LIN {X 0,Y 397.717,Z 584.928,A -85,B 0,C 180,E1 -19257.729,E2 -19257.729} C_VEL
LIN {X 0,Y 395.996,Z 592.127,A -85,B 0,C 180,E1 -19259.493,E2 -19259.493} C_VEL
LIN {X 0,Y 394.774,Z 597.161,A -85,B 0,C 180,E1 -19261.017,E2 -19261.017} C_VEL
LIN {X 0,Y 393.567,Z 602.32,A -85,B 0,C 180,E1 -19263.061,E2 -19263.061} C_VEL
LIN {X 0,Y 392.834,Z 605.925,A -85,B 0,C 180,E1 -19265.115,E2 -19265.115} C_VEL
LIN {X 0,Y 392.166,Z 608.094,A -85,B 0,C 180,E1 -19267.182,E2 -19267.182} C_VEL
LIN {X 0,Y 391.836,Z 608.822,A -85,B 0,C 180,E1 -19269.258,E2 -19269.258} C_VEL
LIN {X 0,Y 391.759,Z 608.57,A -85,B 0,C 180,E1 -19270.455,E2 -19270.455} C_VEL
LIN {X 0,Y 391.593,Z 607.122,A -85,B 0,C 180,E1 -19272.395,E2 -19272.395} C_VEL
LIN {X 0,Y 391.705,Z 604.06,A -85,B 0,C 180,E1 -19274.498,E2 -19274.498} C_VEL
LIN {X 0,Y 391.827,Z 600.696,A -85,B 0,C 180,E1 -19276.086,E2 -19276.086} C_VEL
LIN {X 0,Y 392.017,Z 596.311,A -85,B 0,C 180,E1 -19277.683,E2 -19277.683} C_VEL
LIN {X 0,Y 392.321,Z 589.701,A -85,B 0,C 180,E1 -19279.558,E2 -19279.558} C_VEL
LIN {X 0,Y 392.753,Z 582.648,A -85,B 0,C 180,E1 -19281.17,E2 -19281.17} C_VEL
LIN {X 0,Y 393.306,Z 574.032,A -85,B 0,C 180,E1 -19282.789,E2 -19282.789} C_VEL
LIN {X 0,Y 394.075,Z 563.557,A -85,B 0,C 180,E1 -19284.406,E2 -19284.406} C_VEL
LIN {X 0,Y 394.825,Z 552.905,A -85,B 0,C 180,E1 -19285.763,E2 -19285.763} C_VEL
LIN {X 0,Y 395.691,Z 541.405,A -85,B 0,C 180,E1 -19286.975,E2 -19286.975} C_VEL
LIN {X 0,Y 396.569,Z 527.738,A -85,B 0,C 180,E1 -19288.141,E2 -19288.141} C_VEL
LIN {X 0,Y 397.394,Z 514.095,A -85,B 0,C 180,E1 -19289.066,E2 -19289.066} C_VEL
LIN {X 0,Y 398.175,Z 500.064,A -85,B 0,C 180,E1 -19289.799,E2 -19289.799} C_VEL
LIN {X 0,Y 398.925,Z 485.084,A -85,B 0,C 180,E1 -19290.355,E2 -19290.355} C_VEL
LIN {X 0,Y 400.788,Z 412.237,A -85,B 0,C 180,E1 -19292.1,E2 -19292.1} C_VEL
LIN {X 0,Y 401.807,Z 378.965,A -85,B 0,C 180,E1 -19292.889,E2 -19292.889} C_VEL
LIN {X 0,Y 397.729,Z 345.32,A -85,B 0,C 180,E1 -19293.857,E2 -19293.857} C_VEL
LIN {X 0,Y 397.72,Z 344.139,A -85,B 0,C 180,E1 -19293.988,E2 -19293.988} C_VEL
LIN {X 0,Y 398.553,Z 329.713,A -85,B 0,C 180,E1 -19296.319,E2 -19296.319} C_VEL
LIN {X 0,Y 395.358,Z 313.634,A -85,B 0,C 180,E1 -19299.097,E2 -19299.097} C_VEL
LIN {X 0,Y 394.215,Z 307.939,A -85,B 0,C 180,E1 -19300.103,E2 -19300.103} C_VEL
LIN {X 0,Y 394.182,Z 307.94,A -85,B 0,C 180,E1 -19303.869,E2 -19303.869} C_VEL
LIN {X 0,Y 394.119,Z 307.946,A -85,B 0,C 180,E1 -19307.516,E2 -19307.516} C_VEL
LIN {X 0,Y 394.135,Z 307.949,A -85,B 0,C 180,E1 -19310.222,E2 -19310.222} C_VEL
LIN {X 0,Y 394.157,Z 307.941,A -85,B 0,C 180,E1 -19313.1,E2 -19313.1} C_VEL
LIN {X 0,Y 394.182,Z 307.939,A -85,B 0,C 180,E1 -19316.572,E2 -19316.572} C_VEL
LIN {X 0,Y 394.175,Z 307.944,A -85,B 0,C 180,E1 -19320.159,E2 -19320.159} C_VEL
LIN {X 0,Y 394.204,Z 307.936,A -85,B 0,C 180,E1 -19323.625,E2 -19323.625} C_VEL
LIN {X 0,Y 394.26,Z 307.93,A -85,B 0,C 180,E1 -19327.493,E2 -19327.493} C_VEL
LIN {X 0,Y 394.254,Z 307.93,A -85,B 0,C 180,E1 -19331.347,E2 -19331.347} C_VEL
LIN {X 0,Y 394.308,Z 307.924,A -85,B 0,C 180,E1 -19334.544,E2 -19334.544} C_VEL
LIN {X 0,Y 394.417,Z 307.915,A -85,B 0,C 180,E1 -19337.693,E2 -19337.693} C_VEL
LIN {X 0,Y 394.399,Z 308.039,A -85,B 0,C 180,E1 -19338.871,E2 -19338.871} C_VEL
LIN {X 0,Y 394.702,Z 309.634,A -85,B 0,C 180,E1 -19339.279,E2 -19339.279} C_VEL
LIN {X 0,Y 403.21,Z 335.163,A -85,B 0,C 180,E1 -19340.175,E2 -19340.175} C_VEL
LIN {X 0,Y 403.99,Z 339.498,A -85,B 0,C 180,E1 -19340.292,E2 -19340.292} C_VEL
LIN {X 0,Y 401.838,Z 445.209,A -85,B 0,C 180,E1 -19342.171,E2 -19342.171} C_VEL
LIN {X 0,Y 401.351,Z 459.684,A -85,B 0,C 180,E1 -19342.634,E2 -19342.634} C_VEL
LIN {X 0,Y 400.697,Z 473.526,A -85,B 0,C 180,E1 -19343.284,E2 -19343.284} C_VEL
LIN {X 0,Y 399.792,Z 486.451,A -85,B 0,C 180,E1 -19344.09,E2 -19344.09} C_VEL
LIN {X 0,Y 398.99,Z 497.538,A -85,B 0,C 180,E1 -19344.962,E2 -19344.962} C_VEL
LIN {X 0,Y 397.656,Z 509.289,A -85,B 0,C 180,E1 -19346.084,E2 -19346.084} C_VEL
LIN {X 0,Y 396.813,Z 518.984,A -85,B 0,C 180,E1 -19347.215,E2 -19347.215} C_VEL
LIN {X 0,Y 395.904,Z 528.108,A -85,B 0,C 180,E1 -19348.477,E2 -19348.477} C_VEL
LIN {X 0,Y 394.823,Z 537.282,A -85,B 0,C 180,E1 -19349.998,E2 -19349.998} C_VEL
LIN {X 0,Y 394.061,Z 544.913,A -85,B 0,C 180,E1 -19351.525,E2 -19351.525} C_VEL
LIN {X 0,Y 393.463,Z 551.26,A -85,B 0,C 180,E1 -19353.059,E2 -19353.059} C_VEL
LIN {X 0,Y 393.104,Z 556.487,A -85,B 0,C 180,E1 -19354.596,E2 -19354.596} C_VEL
LIN {X 0,Y 392.549,Z 562.047,A -85,B 0,C 180,E1 -19356.658,E2 -19356.658} C_VEL
LIN {X 0,Y 392.238,Z 565.16,A -85,B 0,C 180,E1 -19358.211,E2 -19358.211} C_VEL
LIN {X 0,Y 392.167,Z 568.068,A -85,B 0,C 180,E1 -19360.286,E2 -19360.286} C_VEL
LIN {X 0,Y 392.135,Z 569.619,A -85,B 0,C 180,E1 -19362.375,E2 -19362.375} C_VEL
LIN {X 0,Y 392.357,Z 569.815,A -85,B 0,C 180,E1 -19364.471,E2 -19364.471} C_VEL
LIN {X 0,Y 392.721,Z 568.654,A -85,B 0,C 180,E1 -19366.578,E2 -19366.578} C_VEL
LIN {X 0,Y 393.38,Z 566.06,A -85,B 0,C 180,E1 -19368.69,E2 -19368.69} C_VEL
LIN {X 0,Y 394.327,Z 561.953,A -85,B 0,C 180,E1 -19370.806,E2 -19370.806} C_VEL
LIN {X 0,Y 395.598,Z 556.204,A -85,B 0,C 180,E1 -19372.922,E2 -19372.922} C_VEL
LIN {X 0,Y 397.028,Z 549.645,A -85,B 0,C 180,E1 -19374.768,E2 -19374.768} C_VEL
LIN {X 0,Y 398.559,Z 542.753,A -85,B 0,C 180,E1 -19376.325,E2 -19376.325} C_VEL
LIN {X 0,Y 400.232,Z 534.249,A -85,B 0,C 180,E1 -19377.911,E2 -19377.911} C_VEL
LIN {X 0,Y 402.147,Z 524.22,A -85,B 0,C 180,E1 -19379.439,E2 -19379.439} C_VEL
LIN {X 0,Y 403.955,Z 513.61,A -85,B 0,C 180,E1 -19380.762,E2 -19380.762} C_VEL
LIN {X 0,Y 405.704,Z 502.263,A -85,B 0,C 180,E1 -19381.917,E2 -19381.917} C_VEL
LIN {X 0,Y 407.33,Z 489.783,A -85,B 0,C 180,E1 -19382.94,E2 -19382.94} C_VEL
LIN {X 0,Y 408.67,Z 476.909,A -85,B 0,C 180,E1 -19383.774,E2 -19383.774} C_VEL
LIN {X 0,Y 409.658,Z 464.519,A -85,B 0,C 180,E1 -19384.393,E2 -19384.393} C_VEL
LIN {X 0,Y 409.957,Z 460.294,A -85,B 0,C 180,E1 -19384.563,E2 -19384.563} C_VEL
LIN {X 0,Y 409.856,Z 454.652,A -85,B 0,C 180,E1 -19384.802,E2 -19384.802} C_VEL
LIN {X 0,Y 407.721,Z 445.503,A -85,B 0,C 180,E1 -19385.244,E2 -19385.244} C_VEL
LIN {X 0,Y 405.273,Z 436.264,A -85,B 0,C 180,E1 -19385.632,E2 -19385.632} C_VEL
LIN {X 0,Y 404.725,Z 430.471,A -85,B 0,C 180,E1 -19385.789,E2 -19385.789} C_VEL
LIN {X 0,Y 407.027,Z 352.192,A -85,B 0,C 180,E1 -19387.172,E2 -19387.172} C_VEL
LIN {X 0,Y 399.145,Z 334.318,A -85,B 0,C 180,E1 -19388.191,E2 -19388.191} C_VEL
LIN {X 0,Y 390.851,Z 317.809,A -85,B 0,C 180,E1 -19389.271,E2 -19389.271} C_VEL
LIN {X 0,Y 387.76,Z 311.713,A -85,B 0,C 180,E1 -19389.72,E2 -19389.72} C_VEL
LIN {X 0,Y 387.081,Z 308.822,A -85,B 0,C 180,E1 -19390.646,E2 -19390.646} C_VEL
LIN {X 0,Y 387.096,Z 308.822,A -85,B 0,C 180,E1 -19393.631,E2 -19393.631} C_VEL
LIN {X 0,Y 387.087,Z 308.827,A -85,B 0,C 180,E1 -19396.558,E2 -19396.558} C_VEL
LIN {X 0,Y 387.084,Z 308.827,A -85,B 0,C 180,E1 -19399.46,E2 -19399.46} C_VEL
LIN {X 0,Y 387.129,Z 308.809,A -85,B 0,C 180,E1 -19402.754,E2 -19402.754} C_VEL
LIN {X 0,Y 387.132,Z 308.804,A -85,B 0,C 180,E1 -19405.883,E2 -19405.883} C_VEL
LIN {X 0,Y 387.133,Z 308.813,A -85,B 0,C 180,E1 -19409.562,E2 -19409.562} C_VEL
LIN {X 0,Y 387.145,Z 308.807,A -85,B 0,C 180,E1 -19413.108,E2 -19413.108} C_VEL
LIN {X 0,Y 387.133,Z 308.818,A -85,B 0,C 180,E1 -19415.409,E2 -19415.409} C_VEL
LIN {X 0,Y 387.191,Z 308.806,A -85,B 0,C 180,E1 -19417.673,E2 -19417.673} C_VEL
LIN {X 0,Y 387.177,Z 308.802,A -85,B 0,C 180,E1 -19420.996,E2 -19420.996} C_VEL
LIN {X 0,Y 387.194,Z 308.809,A -85,B 0,C 180,E1 -19424.255,E2 -19424.255} C_VEL
LIN {X 0,Y 387.311,Z 308.795,A -85,B 0,C 180,E1 -19427.559,E2 -19427.559} C_VEL
LIN {X 0,Y 387.371,Z 308.778,A -85,B 0,C 180,E1 -19431.683,E2 -19431.683} C_VEL
LIN {X 0,Y 387.458,Z 308.776,A -85,B 0,C 180,E1 -19434.814,E2 -19434.814} C_VEL
LIN {X 0,Y 387.4,Z 308.783,A -85,B 0,C 180,E1 -19437.928,E2 -19437.928} C_VEL
LIN {X 0,Y 387.389,Z 308.774,A -85,B 0,C 180,E1 -19441.036,E2 -19441.036} C_VEL
LIN {X 0,Y 387.498,Z 308.771,A -85,B 0,C 180,E1 -19444.146,E2 -19444.146} C_VEL
LIN {X 0,Y 387.402,Z 308.768,A -85,B 0,C 180,E1 -19447.271,E2 -19447.271} C_VEL
LIN {X 0,Y 387.311,Z 308.795,A -85,B 0,C 180,E1 -19450.419,E2 -19450.419} C_VEL
LIN {X 0,Y 387.345,Z 308.775,A -85,B 0,C 180,E1 -19452.533,E2 -19452.533} C_VEL
LIN {X 0,Y 387.248,Z 308.794,A -85,B 0,C 180,E1 -19456.546,E2 -19456.546} C_VEL
LIN {X 0,Y 387.191,Z 308.81,A -85,B 0,C 180,E1 -19460.104,E2 -19460.104} C_VEL
LIN {X 0,Y 387.144,Z 308.815,A -85,B 0,C 180,E1 -19463.456,E2 -19463.456} C_VEL
LIN {X 0,Y 387.145,Z 308.812,A -85,B 0,C 180,E1 -19465.736,E2 -19465.736} C_VEL
LIN {X 0,Y 387.15,Z 308.814,A -85,B 0,C 180,E1 -19469.242,E2 -19469.242} C_VEL
LIN {X 0,Y 387.132,Z 308.817,A -85,B 0,C 180,E1 -19472.874,E2 -19472.874} C_VEL
LIN {X 0,Y 387.198,Z 308.781,A -85,B 0,C 180,E1 -19476.654,E2 -19476.654} C_VEL
LIN {X 0,Y 387.15,Z 308.816,A -85,B 0,C 180,E1 -19479.289,E2 -19479.289} C_VEL
LIN {X 0,Y 387.107,Z 308.823,A -85,B 0,C 180,E1 -19482.114,E2 -19482.114} C_VEL
LIN {X 0,Y 387.143,Z 308.813,A -85,B 0,C 180,E1 -19485.125,E2 -19485.125} C_VEL
LIN {X 0,Y 387.139,Z 308.818,A -85,B 0,C 180,E1 -19487.981,E2 -19487.981} C_VEL
LIN {X 0,Y 387.163,Z 308.815,A -85,B 0,C 180,E1 -19491.073,E2 -19491.073} C_VEL
LIN {X 0,Y 387.226,Z 308.853,A -85,B 0,C 180,E1 -19493.089,E2 -19493.089} C_VEL
LIN {X 0,Y 390.309,Z 320.663,A -85,B 0,C 180,E1 -19496.202,E2 -19496.202} C_VEL
LIN {X 0,Y 392.504,Z 330.055,A -85,B 0,C 180,E1 -19498.538,E2 -19498.538} C_VEL
LIN {X 0,Y 395.104,Z 342.29,A -85,B 0,C 180,E1 -19501.406,E2 -19501.406} C_VEL
LIN {X 0,Y 395.811,Z 345.929,A -85,B 0,C 180,E1 -19502.23,E2 -19502.23} C_VEL
LIN {X 0,Y 395.398,Z 349.986,A -85,B 0,C 180,E1 -19503.051,E2 -19503.051} C_VEL
LIN {X 0,Y 401.869,Z 383.713,A -85,B 0,C 180,E1 -19504.294,E2 -19504.294} C_VEL
LIN {X 0,Y 405.569,Z 408.629,A -85,B 0,C 180,E1 -19505.089,E2 -19505.089} C_VEL
LIN {X 0,Y 403.302,Z 488.379,A -85,B 0,C 180,E1 -19506.527,E2 -19506.527} C_VEL
LIN {X 0,Y 402.306,Z 502.975,A -85,B 0,C 180,E1 -19506.974,E2 -19506.974} C_VEL
LIN {X 0,Y 400.773,Z 516.935,A -85,B 0,C 180,E1 -19507.593,E2 -19507.593} C_VEL
LIN {X 0,Y 399.336,Z 528.164,A -85,B 0,C 180,E1 -19508.254,E2 -19508.254} C_VEL
LIN {X 0,Y 397.405,Z 540.887,A -85,B 0,C 180,E1 -19509.207,E2 -19509.207} C_VEL
LIN {X 0,Y 395.458,Z 552.842,A -85,B 0,C 180,E1 -19510.337,E2 -19510.337} C_VEL
LIN {X 0,Y 393.385,Z 563.621,A -85,B 0,C 180,E1 -19511.579,E2 -19511.579} C_VEL
LIN {X 0,Y 391.238,Z 574.311,A -85,B 0,C 180,E1 -19513.089,E2 -19513.089} C_VEL
LIN {X 0,Y 389.501,Z 583.171,A -85,B 0,C 180,E1 -19514.621,E2 -19514.621} C_VEL
LIN {X 0,Y 387.915,Z 591.702,A -85,B 0,C 180,E1 -19516.427,E2 -19516.427} C_VEL
LIN {X 0,Y 386.65,Z 598.451,A -85,B 0,C 180,E1 -19518.196,E2 -19518.196} C_VEL
LIN {X 0,Y 385.7,Z 604.145,A -85,B 0,C 180,E1 -19520.068,E2 -19520.068} C_VEL
LIN {X 0,Y 385.045,Z 608.993,A -85,B 0,C 180,E1 -19522.161,E2 -19522.161} C_VEL
LIN {X 0,Y 384.927,Z 612.688,A -85,B 0,C 180,E1 -19524.521,E2 -19524.521} C_VEL
LIN {X 0,Y 384.895,Z 613.051,A -85,B 0,C 180,E1 -19524.782,E2 -19524.782} C_VEL
LIN {X 0,Y 384.85,Z 617.082,A -85,B 0,C 180,E1 -19526.35,E2 -19526.35} C_VEL
LIN {X 0,Y 384.85,Z 620.126,A -85,B 0,C 180,E1 -19527.916,E2 -19527.916} C_VEL
LIN {X 0,Y 384.897,Z 621.672,A -85,B 0,C 180,E1 -19528.96,E2 -19528.96} C_VEL
LIN {X 0,Y 384.811,Z 623.592,A -85,B 0,C 180,E1 -19531.045,E2 -19531.045} C_VEL
LIN {X 0,Y 384.734,Z 624.032,A -85,B 0,C 180,E1 -19533.133,E2 -19533.133} C_VEL
LIN {X 0,Y 384.873,Z 623.036,A -85,B 0,C 180,E1 -19535.223,E2 -19535.223} C_VEL
LIN {X 0,Y 385.213,Z 620.617,A -85,B 0,C 180,E1 -19537.315,E2 -19537.315} C_VEL
LIN {X 0,Y 385.94,Z 616.726,A -85,B 0,C 180,E1 -19539.403,E2 -19539.403} C_VEL
LIN {X 0,Y 387.261,Z 611.271,A -85,B 0,C 180,E1 -19541.478,E2 -19541.478} C_VEL
LIN {X 0,Y 388.362,Z 605.739,A -85,B 0,C 180,E1 -19543.11,E2 -19543.11} C_VEL
LIN {X 0,Y 390.047,Z 598.548,A -85,B 0,C 180,E1 -19544.829,E2 -19544.829} C_VEL
LIN {X 0,Y 392.246,Z 589.302,A -85,B 0,C 180,E1 -19546.604,E2 -19546.604} C_VEL
LIN {X 0,Y 394.204,Z 579.747,A -85,B 0,C 180,E1 -19548.119,E2 -19548.119} C_VEL
LIN {X 0,Y 396.511,Z 569.228,A -85,B 0,C 180,E1 -19549.479,E2 -19549.479} C_VEL
LIN {X 0,Y 398.985,Z 556.544,A -85,B 0,C 180,E1 -19550.826,E2 -19550.826} C_VEL
LIN {X 0,Y 401.271,Z 543.87,A -85,B 0,C 180,E1 -19551.91,E2 -19551.91} C_VEL
LIN {X 0,Y 403.32,Z 530.585,A -85,B 0,C 180,E1 -19552.812,E2 -19552.812} C_VEL
LIN {X 0,Y 405.461,Z 514.876,A -85,B 0,C 180,E1 -19553.616,E2 -19553.616} C_VEL
LIN {X 0,Y 407.077,Z 500.015,A -85,B 0,C 180,E1 -19554.157,E2 -19554.157} C_VEL
LIN {X 0,Y 413.308,Z 410.128,A -85,B 0,C 180,E1 -19556.57,E2 -19556.57} C_VEL
LIN {X 0,Y 412.123,Z 392.284,A -85,B 0,C 180,E1 -19557.379,E2 -19557.379} C_VEL
LIN {X 0,Y 410.315,Z 375.608,A -85,B 0,C 180,E1 -19558.261,E2 -19558.261} C_VEL
LIN {X 0,Y 407.875,Z 359.524,A -85,B 0,C 180,E1 -19559.257,E2 -19559.257} C_VEL
LIN {X 0,Y 406.787,Z 354.086,A -85,B 0,C 180,E1 -19559.649,E2 -19559.649} C_VEL
LIN {X 0,Y 405.35,Z 347.684,A -85,B 0,C 180,E1 -19560.497,E2 -19560.497} C_VEL
LIN {X 0,Y 403.914,Z 340.609,A -85,B 0,C 180,E1 -19561.527,E2 -19561.527} C_VEL
LIN {X 0,Y 402.643,Z 336.786,A -85,B 0,C 180,E1 -19562.224,E2 -19562.224} C_VEL
LIN {X 0,Y 398.176,Z 328.661,A -85,B 0,C 180,E1 -19564.26,E2 -19564.26} C_VEL
LIN {X 0,Y 394.492,Z 322.113,A -85,B 0,C 180,E1 -19566.247,E2 -19566.247} C_VEL
LIN {X 0,Y 392.786,Z 318.98,A -85,B 0,C 180,E1 -19567.326,E2 -19567.326} C_VEL
LIN {X 0,Y 390.499,Z 315.506,A -85,B 0,C 180,E1 -19568.891,E2 -19568.891} C_VEL
LIN {X 0,Y 389.955,Z 313.964,A -85,B 0,C 180,E1 -19569.432,E2 -19569.432} C_VEL
LIN {X 0,Y 387.569,Z 310.664,A -85,B 0,C 180,E1 -19571.409,E2 -19571.409} C_VEL
LIN {X 0,Y 387.099,Z 308.821,A -85,B 0,C 180,E1 -19572.381,E2 -19572.381} C_VEL
LIN {X 0,Y 387.121,Z 308.818,A -85,B 0,C 180,E1 -19575.117,E2 -19575.117} C_VEL
LIN {X 0,Y 387.098,Z 308.823,A -85,B 0,C 180,E1 -19577.971,E2 -19577.971} C_VEL
LIN {X 0,Y 387.11,Z 308.823,A -85,B 0,C 180,E1 -19581.085,E2 -19581.085} C_VEL
LIN {X 0,Y 387.174,Z 308.813,A -85,B 0,C 180,E1 -19584.625,E2 -19584.625} C_VEL
LIN {X 0,Y 387.147,Z 308.831,A -85,B 0,C 180,E1 -19586.733,E2 -19586.733} C_VEL
LIN {X 0,Y 388.13,Z 311.639,A -85,B 0,C 180,E1 -19588.443,E2 -19588.443} C_VEL
LIN {X 0,Y 389.475,Z 313.721,A -85,B 0,C 180,E1 -19589.764,E2 -19589.764} C_VEL
LIN {X 0,Y 391.233,Z 317.506,A -85,B 0,C 180,E1 -19591.647,E2 -19591.647} C_VEL
LIN {X 0,Y 393.675,Z 323.256,A -85,B 0,C 180,E1 -19594.046,E2 -19594.046} C_VEL
LIN {X 0,Y 396.597,Z 330.734,A -85,B 0,C 180,E1 -19596.696,E2 -19596.696} C_VEL
LIN {X 0,Y 398.941,Z 337.757,A -85,B 0,C 180,E1 -19598.849,E2 -19598.849} C_VEL
LIN {X 0,Y 401.343,Z 346.482,A -85,B 0,C 180,E1 -19601.22,E2 -19601.22} C_VEL
LIN {X 0,Y 401.755,Z 348.046,A -85,B 0,C 180,E1 -19601.562,E2 -19601.562} C_VEL
LIN {X 0,Y 407.126,Z 358.325,A -85,B 0,C 180,E1 -19602.857,E2 -19602.857} C_VEL
LIN {X 0,Y 410.673,Z 366.267,A -85,B 0,C 180,E1 -19603.695,E2 -19603.695} C_VEL
LIN {X 0,Y 413.329,Z 380.205,A -85,B 0,C 180,E1 -19604.595,E2 -19604.595} C_VEL
LIN {X 0,Y 414.901,Z 391.129,A -85,B 0,C 180,E1 -19605.201,E2 -19605.201} C_VEL
LIN {X 0,Y 407.833,Z 488.797,A -85,B 0,C 180,E1 -19607.792,E2 -19607.792} C_VEL
LIN {X 0,Y 406.346,Z 503.456,A -85,B 0,C 180,E1 -19608.377,E2 -19608.377} C_VEL
LIN {X 0,Y 404.584,Z 517.538,A -85,B 0,C 180,E1 -19609.148,E2 -19609.148} C_VEL
LIN {X 0,Y 402.459,Z 531.281,A -85,B 0,C 180,E1 -19610.104,E2 -19610.104} C_VEL
LIN {X 0,Y 400.294,Z 543.672,A -85,B 0,C 180,E1 -19611.193,E2 -19611.193} C_VEL
LIN {X 0,Y 397.851,Z 556.012,A -85,B 0,C 180,E1 -19612.539,E2 -19612.539} C_VEL
LIN {X 0,Y 395.719,Z 566.254,A -85,B 0,C 180,E1 -19613.903,E2 -19613.903} C_VEL
LIN {X 0,Y 393.861,Z 574.529,A -85,B 0,C 180,E1 -19615.221,E2 -19615.221} C_VEL
LIN {X 0,Y 391.606,Z 583.459,A -85,B 0,C 180,E1 -19616.924,E2 -19616.924} C_VEL
LIN {X 0,Y 389.876,Z 590.014,A -85,B 0,C 180,E1 -19618.456,E2 -19618.456} C_VEL
LIN {X 0,Y 388.079,Z 597.03,A -85,B 0,C 180,E1 -19620.517,E2 -19620.517} C_VEL
LIN {X 0,Y 387.039,Z 601.106,A -85,B 0,C 180,E1 -19622.074,E2 -19622.074} C_VEL
LIN {X 0,Y 386.112,Z 605.178,A -85,B 0,C 180,E1 -19624.161,E2 -19624.161} C_VEL
LIN {X 0,Y 385.351,Z 607.788,A -85,B 0,C 180,E1 -19626.261,E2 -19626.261} C_VEL
LIN {X 0,Y 384.833,Z 608.92,A -85,B 0,C 180,E1 -19628.373,E2 -19628.373} C_VEL
LIN {X 0,Y 384.652,Z 608.602,A -85,B 0,C 180,E1 -19630.492,E2 -19630.492} C_VEL
LIN {X 0,Y 384.504,Z 606.802,A -85,B 0,C 180,E1 -19632.627,E2 -19632.627} C_VEL
LIN {X 0,Y 384.627,Z 603.466,A -85,B 0,C 180,E1 -19634.771,E2 -19634.771} C_VEL
LIN {X 0,Y 384.772,Z 599.82,A -85,B 0,C 180,E1 -19636.389,E2 -19636.389} C_VEL
LIN {X 0,Y 384.97,Z 595.132,A -85,B 0,C 180,E1 -19638.018,E2 -19638.018} C_VEL
LIN {X 0,Y 385.334,Z 588.18,A -85,B 0,C 180,E1 -19639.927,E2 -19639.927} C_VEL
LIN {X 0,Y 385.755,Z 580.768,A -85,B 0,C 180,E1 -19641.568,E2 -19641.568} C_VEL
LIN {X 0,Y 386.378,Z 571.701,A -85,B 0,C 180,E1 -19643.222,E2 -19643.222} C_VEL
LIN {X 0,Y 387.175,Z 561.079,A -85,B 0,C 180,E1 -19644.806,E2 -19644.806} C_VEL
LIN {X 0,Y 388.055,Z 549.327,A -85,B 0,C 180,E1 -19646.246,E2 -19646.246} C_VEL
LIN {X 0,Y 388.918,Z 537.005,A -85,B 0,C 180,E1 -19647.484,E2 -19647.484} C_VEL
LIN {X 0,Y 389.774,Z 524.543,A -85,B 0,C 180,E1 -19648.504,E2 -19648.504} C_VEL
LIN {X 0,Y 390.571,Z 510.645,A -85,B 0,C 180,E1 -19649.402,E2 -19649.402} C_VEL
LIN {X 0,Y 391.353,Z 495.282,A -85,B 0,C 180,E1 -19650.15,E2 -19650.15} C_VEL
LIN {X 0,Y 391.98,Z 480.362,A -85,B 0,C 180,E1 -19650.653,E2 -19650.653} C_VEL
LIN {X 0,Y 394.773,Z 379.081,A -85,B 0,C 180,E1 -19653.104,E2 -19653.104} C_VEL
LIN {X 0,Y 390.726,Z 344.841,A -85,B 0,C 180,E1 -19654.132,E2 -19654.132} C_VEL
LIN {X 0,Y 391.585,Z 330.973,A -85,B 0,C 180,E1 -19656.393,E2 -19656.393} C_VEL
LIN {X 0,Y 388.442,Z 315.155,A -85,B 0,C 180,E1 -19659.158,E2 -19659.158} C_VEL
LIN {X 0,Y 387.138,Z 308.822,A -85,B 0,C 180,E1 -19660.292,E2 -19660.292} C_VEL
LIN {X 0,Y 387.119,Z 308.819,A -85,B 0,C 180,E1 -19663.632,E2 -19663.632} C_VEL
LIN {X 0,Y 387.083,Z 308.827,A -85,B 0,C 180,E1 -19666.555,E2 -19666.555} C_VEL
LIN {X 0,Y 387.096,Z 308.82,A -85,B 0,C 180,E1 -19669.463,E2 -19669.463} C_VEL
LIN {X 0,Y 387.131,Z 308.818,A -85,B 0,C 180,E1 -19672.759,E2 -19672.759} C_VEL
LIN {X 0,Y 387.118,Z 308.819,A -85,B 0,C 180,E1 -19676.337,E2 -19676.337} C_VEL
LIN {X 0,Y 387.126,Z 308.818,A -85,B 0,C 180,E1 -19679.559,E2 -19679.559} C_VEL
LIN {X 0,Y 387.154,Z 308.812,A -85,B 0,C 180,E1 -19683.106,E2 -19683.106} C_VEL
LIN {X 0,Y 387.14,Z 308.816,A -85,B 0,C 180,E1 -19685.407,E2 -19685.407} C_VEL
LIN {X 0,Y 387.218,Z 308.809,A -85,B 0,C 180,E1 -19687.672,E2 -19687.672} C_VEL
LIN {X 0,Y 387.208,Z 308.807,A -85,B 0,C 180,E1 -19690.995,E2 -19690.995} C_VEL
LIN {X 0,Y 387.267,Z 308.804,A -85,B 0,C 180,E1 -19694.256,E2 -19694.256} C_VEL
LIN {X 0,Y 387.34,Z 308.796,A -85,B 0,C 180,E1 -19697.556,E2 -19697.556} C_VEL
LIN {X 0,Y 387.357,Z 308.885,A -85,B 0,C 180,E1 -19698.623,E2 -19698.623} C_VEL
LIN {X 0,Y 387.566,Z 310.046,A -85,B 0,C 180,E1 -19698.924,E2 -19698.924} C_VEL
LIN {X 0,Y 396.649,Z 337.095,A -85,B 0,C 180,E1 -19699.9,E2 -19699.9} C_VEL
LIN {X 0,Y 397.206,Z 339.535,A -85,B 0,C 180,E1 -19699.972,E2 -19699.972} C_VEL
LIN {X 0,Y 395.021,Z 446.166,A -85,B 0,C 180,E1 -19701.907,E2 -19701.907} C_VEL
LIN {X 0,Y 394.514,Z 460.458,A -85,B 0,C 180,E1 -19702.377,E2 -19702.377} C_VEL
LIN {X 0,Y 393.847,Z 474.202,A -85,B 0,C 180,E1 -19703.039,E2 -19703.039} C_VEL
LIN {X 0,Y 392.91,Z 487.072,A -85,B 0,C 180,E1 -19703.857,E2 -19703.857} C_VEL
LIN {X 0,Y 392.048,Z 498.129,A -85,B 0,C 180,E1 -19704.744,E2 -19704.744} C_VEL
LIN {X 0,Y 390.731,Z 509.837,A -85,B 0,C 180,E1 -19705.886,E2 -19705.886} C_VEL
LIN {X 0,Y 389.786,Z 520.471,A -85,B 0,C 180,E1 -19707.165,E2 -19707.165} C_VEL
LIN {X 0,Y 388.804,Z 529.429,A -85,B 0,C 180,E1 -19708.449,E2 -19708.449} C_VEL
LIN {X 0,Y 387.744,Z 538.445,A -85,B 0,C 180,E1 -19709.997,E2 -19709.997} C_VEL
LIN {X 0,Y 386.9,Z 545.956,A -85,B 0,C 180,E1 -19711.554,E2 -19711.554} C_VEL
LIN {X 0,Y 386.398,Z 552.209,A -85,B 0,C 180,E1 -19713.115,E2 -19713.115} C_VEL
LIN {X 0,Y 385.986,Z 557.355,A -85,B 0,C 180,E1 -19714.681,E2 -19714.681} C_VEL
LIN {X 0,Y 385.557,Z 561.561,A -85,B 0,C 180,E1 -19716.255,E2 -19716.255} C_VEL
LIN {X 0,Y 385.143,Z 565.827,A -85,B 0,C 180,E1 -19718.363,E2 -19718.363} C_VEL
LIN {X 0,Y 385.081,Z 568.644,A -85,B 0,C 180,E1 -19720.477,E2 -19720.477} C_VEL
LIN {X 0,Y 385.069,Z 570.106,A -85,B 0,C 180,E1 -19722.605,E2 -19722.605} C_VEL
LIN {X 0,Y 385.304,Z 570.209,A -85,B 0,C 180,E1 -19724.741,E2 -19724.741} C_VEL
LIN {X 0,Y 385.711,Z 568.928,A -85,B 0,C 180,E1 -19726.888,E2 -19726.888} C_VEL
LIN {X 0,Y 386.429,Z 566.227,A -85,B 0,C 180,E1 -19729.04,E2 -19729.04} C_VEL
LIN {X 0,Y 387.474,Z 562.018,A -85,B 0,C 180,E1 -19731.192,E2 -19731.192} C_VEL
LIN {X 0,Y 388.815,Z 556.161,A -85,B 0,C 180,E1 -19733.346,E2 -19733.346} C_VEL
LIN {X 0,Y 390.336,Z 549.486,A -85,B 0,C 180,E1 -19735.222,E2 -19735.222} C_VEL
LIN {X 0,Y 392.156,Z 541.35,A -85,B 0,C 180,E1 -19737.034,E2 -19737.034} C_VEL
LIN {X 0,Y 394.06,Z 532.196,A -85,B 0,C 180,E1 -19738.677,E2 -19738.677} C_VEL
LIN {X 0,Y 396.164,Z 521.352,A -85,B 0,C 180,E1 -19740.254,E2 -19740.254} C_VEL
LIN {X 0,Y 398.065,Z 510.297,A -85,B 0,C 180,E1 -19741.563,E2 -19741.563} C_VEL
LIN {X 0,Y 399.77,Z 499.188,A -85,B 0,C 180,E1 -19742.637,E2 -19742.637} C_VEL
LIN {X 0,Y 401.385,Z 486.322,A -85,B 0,C 180,E1 -19743.642,E2 -19743.642} C_VEL
LIN {X 0,Y 402.69,Z 472.317,A -85,B 0,C 180,E1 -19744.496,E2 -19744.496} C_VEL
LIN {X 0,Y 403.755,Z 458.331,A -85,B 0,C 180,E1 -19745.107,E2 -19745.107} C_VEL
LIN {X 0,Y 404.44,Z 444.533,A -85,B 0,C 180,E1 -19745.513,E2 -19745.513} C_VEL
LIN {X 0,Y 404.725,Z 430.471,A -85,B 0,C 180,E1 -19745.789,E2 -19745.789} C_VEL
LIN {X 0,Y 404.266,Z 424.679,A -85,B 0,C 180,E1 -19745.939,E2 -19745.939} C_VEL
LIN {X 0,Y 399.912,Z 406.019,A -85,B 0,C 180,E1 -19746.658,E2 -19746.658} C_VEL
LIN {X 0,Y 399.426,Z 400.229,A -85,B 0,C 180,E1 -19746.815,E2 -19746.815} C_VEL
LIN {X 0,Y 400.821,Z 354.039,A -85,B 0,C 180,E1 -19747.644,E2 -19747.644} C_VEL
LIN {X 0,Y 393.009,Z 336.465,A -85,B 0,C 180,E1 -19748.68,E2 -19748.68} C_VEL
LIN {X 0,Y 384.345,Z 319.332,A -85,B 0,C 180,E1 -19749.846,E2 -19749.846} C_VEL
LIN {X 0,Y 380.665,Z 312.27,A -85,B 0,C 180,E1 -19750.375,E2 -19750.375} C_VEL
LIN {X 0,Y 380.012,Z 309.697,A -85,B 0,C 180,E1 -19751.232,E2 -19751.232} C_VEL
LIN {X 0,Y 380.054,Z 309.687,A -85,B 0,C 180,E1 -19754.45,E2 -19754.45} C_VEL
LIN {X 0,Y 380.022,Z 309.704,A -85,B 0,C 180,E1 -19757.494,E2 -19757.494} C_VEL
LIN {X 0,Y 380.056,Z 309.701,A -85,B 0,C 180,E1 -19761.199,E2 -19761.199} C_VEL
LIN {X 0,Y 380.082,Z 309.667,A -85,B 0,C 180,E1 -19764.175,E2 -19764.175} C_VEL
LIN {X 0,Y 380.075,Z 309.7,A -85,B 0,C 180,E1 -19767.694,E2 -19767.694} C_VEL
LIN {X 0,Y 380.114,Z 309.693,A -85,B 0,C 180,E1 -19770.163,E2 -19770.163} C_VEL
LIN {X 0,Y 380.093,Z 309.692,A -85,B 0,C 180,E1 -19773.751,E2 -19773.751} C_VEL
LIN {X 0,Y 380.117,Z 309.682,A -85,B 0,C 180,E1 -19777.234,E2 -19777.234} C_VEL
LIN {X 0,Y 380.141,Z 309.68,A -85,B 0,C 180,E1 -19780.63,E2 -19780.63} C_VEL
LIN {X 0,Y 380.157,Z 309.687,A -85,B 0,C 180,E1 -19783.956,E2 -19783.956} C_VEL
LIN {X 0,Y 380.268,Z 309.67,A -85,B 0,C 180,E1 -19787.471,E2 -19787.471} C_VEL
LIN {X 0,Y 380.319,Z 309.655,A -85,B 0,C 180,E1 -19791.527,E2 -19791.527} C_VEL
LIN {X 0,Y 380.409,Z 309.655,A -85,B 0,C 180,E1 -19794.718,E2 -19794.718} C_VEL
LIN {X 0,Y 380.378,Z 309.658,A -85,B 0,C 180,E1 -19797.889,E2 -19797.889} C_VEL
LIN {X 0,Y 380.356,Z 309.649,A -85,B 0,C 180,E1 -19801.055,E2 -19801.055} C_VEL
LIN {X 0,Y 380.467,Z 309.647,A -85,B 0,C 180,E1 -19804.223,E2 -19804.223} C_VEL
LIN {X 0,Y 380.357,Z 309.645,A -85,B 0,C 180,E1 -19807.407,E2 -19807.407} C_VEL
LIN {X 0,Y 380.261,Z 309.673,A -85,B 0,C 180,E1 -19810.615,E2 -19810.615} C_VEL
LIN {X 0,Y 380.279,Z 309.655,A -85,B 0,C 180,E1 -19812.77,E2 -19812.77} C_VEL
LIN {X 0,Y 380.204,Z 309.677,A -85,B 0,C 180,E1 -19816.042,E2 -19816.042} C_VEL
LIN {X 0,Y 380.162,Z 309.685,A -85,B 0,C 180,E1 -19820.014,E2 -19820.014} C_VEL
LIN {X 0,Y 380.102,Z 309.692,A -85,B 0,C 180,E1 -19823.917,E2 -19823.917} C_VEL
LIN {X 0,Y 380.126,Z 309.688,A -85,B 0,C 180,E1 -19827.43,E2 -19827.43} C_VEL
LIN {X 0,Y 380.084,Z 309.691,A -85,B 0,C 180,E1 -19831.065,E2 -19831.065} C_VEL
LIN {X 0,Y 380.1,Z 309.664,A -85,B 0,C 180,E1 -19834.839,E2 -19834.839} C_VEL
LIN {X 0,Y 380.164,Z 309.675,A -85,B 0,C 180,E1 -19837.608,E2 -19837.608} C_VEL
LIN {X 0,Y 380.057,Z 309.699,A -85,B 0,C 180,E1 -19840.925,E2 -19840.925} C_VEL
LIN {X 0,Y 380.105,Z 309.694,A -85,B 0,C 180,E1 -19844.447,E2 -19844.447} C_VEL
LIN {X 0,Y 380.085,Z 309.694,A -85,B 0,C 180,E1 -19847.489,E2 -19847.489} C_VEL
LIN {X 0,Y 380.114,Z 309.693,A -85,B 0,C 180,E1 -19851.21,E2 -19851.21} C_VEL
LIN {X 0,Y 380.166,Z 309.778,A -85,B 0,C 180,E1 -19852.492,E2 -19852.492} C_VEL
LIN {X 0,Y 383.099,Z 320.722,A -85,B 0,C 180,E1 -19855.477,E2 -19855.477} C_VEL
LIN {X 0,Y 385.643,Z 331.469,A -85,B 0,C 180,E1 -19858.219,E2 -19858.219} C_VEL
LIN {X 0,Y 388.238,Z 343.647,A -85,B 0,C 180,E1 -19861.148,E2 -19861.148} C_VEL
LIN {X 0,Y 388.994,Z 347.723,A -85,B 0,C 180,E1 -19862.088,E2 -19862.088} C_VEL
LIN {X 0,Y 388.884,Z 349.574,A -85,B 0,C 180,E1 -19862.476,E2 -19862.476} C_VEL
LIN {X 0,Y 395.239,Z 382.327,A -85,B 0,C 180,E1 -19863.718,E2 -19863.718} C_VEL
LIN {X 0,Y 399.251,Z 408.824,A -85,B 0,C 180,E1 -19864.593,E2 -19864.593} C_VEL
LIN {X 0,Y 397.589,Z 469.051,A -85,B 0,C 180,E1 -19865.685,E2 -19865.685} C_VEL
LIN {X 0,Y 396.883,Z 490.656,A -85,B 0,C 180,E1 -19866.124,E2 -19866.124} C_VEL
LIN {X 0,Y 395.732,Z 505.104,A -85,B 0,C 180,E1 -19866.603,E2 -19866.603} C_VEL
LIN {X 0,Y 394.085,Z 518.965,A -85,B 0,C 180,E1 -19867.261,E2 -19867.261} C_VEL
LIN {X 0,Y 392.298,Z 532.21,A -85,B 0,C 180,E1 -19868.114,E2 -19868.114} C_VEL
LIN {X 0,Y 390.529,Z 542.92,A -85,B 0,C 180,E1 -19868.982,E2 -19868.982} C_VEL
LIN {X 0,Y 388.339,Z 555.434,A -85,B 0,C 180,E1 -19870.236,E2 -19870.236} C_VEL
LIN {X 0,Y 386.284,Z 565.708,A -85,B 0,C 180,E1 -19871.502,E2 -19871.502} C_VEL
LIN {X 0,Y 384.091,Z 575.976,A -85,B 0,C 180,E1 -19873.038,E2 -19873.038} C_VEL
LIN {X 0,Y 382.361,Z 584.494,A -85,B 0,C 180,E1 -19874.599,E2 -19874.599} C_VEL
LIN {X 0,Y 380.784,Z 592.684,A -85,B 0,C 180,E1 -19876.439,E2 -19876.439} C_VEL
LIN {X 0,Y 379.489,Z 599.32,A -85,B 0,C 180,E1 -19878.288,E2 -19878.288} C_VEL
LIN {X 0,Y 378.486,Z 605.259,A -85,B 0,C 180,E1 -19880.415,E2 -19880.415} C_VEL
LIN {X 0,Y 377.868,Z 609.658,A -85,B 0,C 180,E1 -19882.547,E2 -19882.547} C_VEL
LIN {X 0,Y 377.812,Z 612.781,A -85,B 0,C 180,E1 -19884.817,E2 -19884.817} C_VEL
LIN {X 0,Y 377.775,Z 617.617,A -85,B 0,C 180,E1 -19886.814,E2 -19886.814} C_VEL
LIN {X 0,Y 377.824,Z 621.235,A -85,B 0,C 180,E1 -19888.94,E2 -19888.94} C_VEL
LIN {X 0,Y 377.735,Z 623.311,A -85,B 0,C 180,E1 -19891.065,E2 -19891.065} C_VEL
LIN {X 0,Y 377.642,Z 623.902,A -85,B 0,C 180,E1 -19893.192,E2 -19893.192} C_VEL
LIN {X 0,Y 377.808,Z 623.036,A -85,B 0,C 180,E1 -19895.321,E2 -19895.321} C_VEL
LIN {X 0,Y 378.144,Z 620.746,A -85,B 0,C 180,E1 -19897.453,E2 -19897.453} C_VEL
LIN {X 0,Y 378.938,Z 617,A -85,B 0,C 180,E1 -19899.579,E2 -19899.579} C_VEL
LIN {X 0,Y 380.303,Z 611.694,A -85,B 0,C 180,E1 -19901.691,E2 -19901.691} C_VEL
LIN {X 0,Y 381.639,Z 605.717,A -85,B 0,C 180,E1 -19903.521,E2 -19903.521} C_VEL
LIN {X 0,Y 383.523,Z 598.161,A -85,B 0,C 180,E1 -19905.359,E2 -19905.359} C_VEL
LIN {X 0,Y 385.825,Z 588.895,A -85,B 0,C 180,E1 -19907.16,E2 -19907.16} C_VEL
LIN {X 0,Y 387.997,Z 579.284,A -85,B 0,C 180,E1 -19908.692,E2 -19908.692} C_VEL
LIN {X 0,Y 390.647,Z 567.715,A -85,B 0,C 180,E1 -19910.194,E2 -19910.194} C_VEL
LIN {X 0,Y 393.021,Z 556.072,A -85,B 0,C 180,E1 -19911.432,E2 -19911.432} C_VEL
LIN {X 0,Y 395.436,Z 543.343,A -85,B 0,C 180,E1 -19912.525,E2 -19912.525} C_VEL
LIN {X 0,Y 397.619,Z 529.775,A -85,B 0,C 180,E1 -19913.453,E2 -19913.453} C_VEL
LIN {X 0,Y 399.69,Z 515.382,A -85,B 0,C 180,E1 -19914.198,E2 -19914.198} C_VEL
LIN {X 0,Y 401.423,Z 500.424,A -85,B 0,C 180,E1 -19914.76,E2 -19914.76} C_VEL
LIN {X 0,Y 407.988,Z 410.901,A -85,B 0,C 180,E1 -19917.219,E2 -19917.219} C_VEL
LIN {X 0,Y 406.824,Z 392.448,A -85,B 0,C 180,E1 -19918.09,E2 -19918.09} C_VEL
LIN {X 0,Y 405.093,Z 376.467,A -85,B 0,C 180,E1 -19918.978,E2 -19918.978} C_VEL
LIN {X 0,Y 403.04,Z 362.154,A -85,B 0,C 180,E1 -19919.894,E2 -19919.894} C_VEL
LIN {X 0,Y 402.103,Z 357.358,A -85,B 0,C 180,E1 -19920.25,E2 -19920.25} C_VEL
LIN {X 0,Y 400.573,Z 352.896,A -85,B 0,C 180,E1 -19920.739,E2 -19920.739} C_VEL
LIN {X 0,Y 398.967,Z 344.76,A -85,B 0,C 180,E1 -19921.943,E2 -19921.943} C_VEL
LIN {X 0,Y 397.596,Z 340.998,A -85,B 0,C 180,E1 -19922.683,E2 -19922.683} C_VEL
LIN {X 0,Y 392.949,Z 332.379,A -85,B 0,C 180,E1 -19924.919,E2 -19924.919} C_VEL
LIN {X 0,Y 388.562,Z 324.541,A -85,B 0,C 180,E1 -19927.517,E2 -19927.517} C_VEL
LIN {X 0,Y 385.898,Z 320.013,A -85,B 0,C 180,E1 -19929.444,E2 -19929.444} C_VEL
LIN {X 0,Y 383.496,Z 316.434,A -85,B 0,C 180,E1 -19931.509,E2 -19931.509} C_VEL
LIN {X 0,Y 382.746,Z 314.404,A -85,B 0,C 180,E1 -19932.621,E2 -19932.621} C_VEL
LIN {X 0,Y 380.509,Z 311.502,A -85,B 0,C 180,E1 -19935.885,E2 -19935.885} C_VEL
LIN {X 0,Y 380.084,Z 310.005,A -85,B 0,C 180,E1 -19938.438,E2 -19938.438} C_VEL
LIN {X 0,Y 380.159,Z 310.2,A -85,B 0,C 180,E1 -19941.211,E2 -19941.211} C_VEL
LIN {X 0,Y 380.809,Z 311.962,A -85,B 0,C 180,E1 -19944.032,E2 -19944.032} C_VEL
LIN {X 0,Y 382.539,Z 314.299,A -85,B 0,C 180,E1 -19946.68,E2 -19946.68} C_VEL
LIN {X 0,Y 384.006,Z 317.872,A -85,B 0,C 180,E1 -19949.018,E2 -19949.018} C_VEL
LIN {X 0,Y 385.974,Z 321.72,A -85,B 0,C 180,E1 -19951.175,E2 -19951.175} C_VEL
LIN {X 0,Y 389.008,Z 329.246,A -85,B 0,C 180,E1 -19954.396,E2 -19954.396} C_VEL
LIN {X 0,Y 391.71,Z 336.672,A -85,B 0,C 180,E1 -19957.02,E2 -19957.02} C_VEL
LIN {X 0,Y 394.165,Z 344.686,A -85,B 0,C 180,E1 -19959.454,E2 -19959.454} C_VEL
LIN {X 0,Y 395.184,Z 348.256,A -85,B 0,C 180,E1 -19960.406,E2 -19960.406} C_VEL
LIN {X 0,Y 401.384,Z 359.916,A -85,B 0,C 180,E1 -19962.018,E2 -19962.018} C_VEL
LIN {X 0,Y 405.848,Z 369.619,A -85,B 0,C 180,E1 -19963.126,E2 -19963.126} C_VEL
LIN {X 0,Y 408.247,Z 382.609,A -85,B 0,C 180,E1 -19963.992,E2 -19963.992} C_VEL
LIN {X 0,Y 409.573,Z 392.898,A -85,B 0,C 180,E1 -19964.572,E2 -19964.572} C_VEL
LIN {X 0,Y 402.187,Z 489.52,A -85,B 0,C 180,E1 -19967.191,E2 -19967.191} C_VEL
LIN {X 0,Y 400.563,Z 504.57,A -85,B 0,C 180,E1 -19967.817,E2 -19967.817} C_VEL
LIN {X 0,Y 398.7,Z 518.549,A -85,B 0,C 180,E1 -19968.601,E2 -19968.601} C_VEL
LIN {X 0,Y 396.496,Z 532.08,A -85,B 0,C 180,E1 -19969.568,E2 -19969.568} C_VEL
LIN {X 0,Y 394.206,Z 544.298,A -85,B 0,C 180,E1 -19970.669,E2 -19970.669} C_VEL
LIN {X 0,Y 391.634,Z 556.578,A -85,B 0,C 180,E1 -19972.033,E2 -19972.033} C_VEL
LIN {X 0,Y 389.213,Z 567.573,A -85,B 0,C 180,E1 -19973.542,E2 -19973.542} C_VEL
LIN {X 0,Y 386.935,Z 577.076,A -85,B 0,C 180,E1 -19975.131,E2 -19975.131} C_VEL
LIN {X 0,Y 384.585,Z 585.581,A -85,B 0,C 180,E1 -19976.868,E2 -19976.868} C_VEL
LIN {X 0,Y 382.845,Z 591.811,A -85,B 0,C 180,E1 -19978.427,E2 -19978.427} C_VEL
LIN {X 0,Y 381.011,Z 598.398,A -85,B 0,C 180,E1 -19980.527,E2 -19980.527} C_VEL
LIN {X 0,Y 379.668,Z 603.314,A -85,B 0,C 180,E1 -19982.644,E2 -19982.644} C_VEL
LIN {X 0,Y 379.011,Z 605.988,A -85,B 0,C 180,E1 -19984.239,E2 -19984.239} C_VEL
LIN {X 0,Y 378.224,Z 608.276,A -85,B 0,C 180,E1 -19986.38,E2 -19986.38} C_VEL
LIN {X 0,Y 377.725,Z 609.135,A -85,B 0,C 180,E1 -19988.531,E2 -19988.531} C_VEL
LIN {X 0,Y 377.545,Z 608.545,A -85,B 0,C 180,E1 -19990.692,E2 -19990.692} C_VEL
LIN {X 0,Y 377.402,Z 606.456,A -85,B 0,C 180,E1 -19992.869,E2 -19992.869} C_VEL
LIN {X 0,Y 377.505,Z 603.835,A -85,B 0,C 180,E1 -19994.506,E2 -19994.506} C_VEL
LIN {X 0,Y 377.648,Z 600.265,A -85,B 0,C 180,E1 -19996.154,E2 -19996.154} C_VEL
LIN {X 0,Y 377.855,Z 595.663,A -85,B 0,C 180,E1 -19997.81,E2 -19997.81} C_VEL
LIN {X 0,Y 378.186,Z 588.806,A -85,B 0,C 180,E1 -19999.756,E2 -19999.756} C_VEL
LIN {X 0,Y 378.622,Z 581.478,A -85,B 0,C 180,E1 -20001.43,E2 -20001.43} C_VEL
LIN {X 0,Y 379.231,Z 572.563,A -85,B 0,C 180,E1 -20003.11,E2 -20003.11} C_VEL
LIN {X 0,Y 379.919,Z 563.64,A -85,B 0,C 180,E1 -20004.508,E2 -20004.508} C_VEL
LIN {X 0,Y 380.744,Z 552.219,A -85,B 0,C 180,E1 -20006.002,E2 -20006.002} C_VEL
LIN {X 0,Y 381.663,Z 539.925,A -85,B 0,C 180,E1 -20007.31,E2 -20007.31} C_VEL
LIN {X 0,Y 382.608,Z 526.055,A -85,B 0,C 180,E1 -20008.506,E2 -20008.506} C_VEL
LIN {X 0,Y 383.396,Z 512.897,A -85,B 0,C 180,E1 -20009.406,E2 -20009.406} C_VEL
LIN {X 0,Y 384.231,Z 498.334,A -85,B 0,C 180,E1 -20010.163,E2 -20010.163} C_VEL
LIN {X 0,Y 384.926,Z 483.218,A -85,B 0,C 180,E1 -20010.72,E2 -20010.72} C_VEL
LIN {X 0,Y 387.836,Z 379.832,A -85,B 0,C 180,E1 -20013.307,E2 -20013.307} C_VEL
LIN {X 0,Y 383.811,Z 345.399,A -85,B 0,C 180,E1 -20014.339,E2 -20014.339} C_VEL
LIN {X 0,Y 384.567,Z 331.841,A -85,B 0,C 180,E1 -20016.539,E2 -20016.539} C_VEL
LIN {X 0,Y 380.777,Z 312.919,A -85,B 0,C 180,E1 -20019.889,E2 -20019.889} C_VEL
LIN {X 0,Y 380.085,Z 309.701,A -85,B 0,C 180,E1 -20020.482,E2 -20020.482} C_VEL
LIN {X 0,Y 380.076,Z 309.698,A -85,B 0,C 180,E1 -20024.451,E2 -20024.451} C_VEL
LIN {X 0,Y 380.019,Z 309.703,A -85,B 0,C 180,E1 -20027.5,E2 -20027.5} C_VEL
LIN {X 0,Y 380.054,Z 309.698,A -85,B 0,C 180,E1 -20031.196,E2 -20031.196} C_VEL
LIN {X 0,Y 380.074,Z 309.699,A -85,B 0,C 180,E1 -20034.182,E2 -20034.182} C_VEL
LIN {X 0,Y 380.05,Z 309.698,A -85,B 0,C 180,E1 -20037.689,E2 -20037.689} C_VEL
LIN {X 0,Y 380.082,Z 309.693,A -85,B 0,C 180,E1 -20041.368,E2 -20041.368} C_VEL
LIN {X 0,Y 380.122,Z 309.692,A -85,B 0,C 180,E1 -20044.544,E2 -20044.544} C_VEL
LIN {X 0,Y 380.134,Z 309.691,A -85,B 0,C 180,E1 -20048.373,E2 -20048.373} C_VEL
LIN {X 0,Y 380.171,Z 309.684,A -85,B 0,C 180,E1 -20050.629,E2 -20050.629} C_VEL
LIN {X 0,Y 380.229,Z 309.682,A -85,B 0,C 180,E1 -20053.957,E2 -20053.957} C_VEL
LIN {X 0,Y 380.296,Z 309.673,A -85,B 0,C 180,E1 -20057.468,E2 -20057.468} C_VEL
LIN {X 0,Y 380.315,Z 309.729,A -85,B 0,C 180,E1 -20058.357,E2 -20058.357} C_VEL
LIN {X 0,Y 380.439,Z 310.438,A -85,B 0,C 180,E1 -20058.544,E2 -20058.544} C_VEL
LIN {X 0,Y 389.352,Z 336.656,A -85,B 0,C 180,E1 -20059.534,E2 -20059.534} C_VEL
LIN {X 0,Y 390.47,Z 340.538,A -85,B 0,C 180,E1 -20059.664,E2 -20059.664} C_VEL
LIN {X 0,Y 388.246,Z 445.991,A -85,B 0,C 180,E1 -20061.601,E2 -20061.601} C_VEL
LIN {X 0,Y 387.722,Z 460.48,A -85,B 0,C 180,E1 -20062.08,E2 -20062.08} C_VEL
LIN {X 0,Y 387.006,Z 474.878,A -85,B 0,C 180,E1 -20062.784,E2 -20062.784} C_VEL
LIN {X 0,Y 386.037,Z 487.692,A -85,B 0,C 180,E1 -20063.617,E2 -20063.617} C_VEL
LIN {X 0,Y 385.121,Z 498.717,A -85,B 0,C 180,E1 -20064.518,E2 -20064.518} C_VEL
LIN {X 0,Y 383.789,Z 510.39,A -85,B 0,C 180,E1 -20065.68,E2 -20065.68} C_VEL
LIN {X 0,Y 382.906,Z 520.035,A -85,B 0,C 180,E1 -20066.852,E2 -20066.852} C_VEL
LIN {X 0,Y 381.923,Z 529.125,A -85,B 0,C 180,E1 -20068.158,E2 -20068.158} C_VEL
LIN {X 0,Y 380.785,Z 538.267,A -85,B 0,C 180,E1 -20069.734,E2 -20069.734} C_VEL
LIN {X 0,Y 379.949,Z 545.875,A -85,B 0,C 180,E1 -20071.318,E2 -20071.318} C_VEL
LIN {X 0,Y 379.397,Z 551.207,A -85,B 0,C 180,E1 -20072.643,E2 -20072.643} C_VEL
LIN {X 0,Y 379.066,Z 556.601,A -85,B 0,C 180,E1 -20074.236,E2 -20074.236} C_VEL
LIN {X 0,Y 378.455,Z 562.323,A -85,B 0,C 180,E1 -20076.373,E2 -20076.373} C_VEL
LIN {X 0,Y 378.056,Z 566.493,A -85,B 0,C 180,E1 -20078.521,E2 -20078.521} C_VEL
LIN {X 0,Y 377.974,Z 569.223,A -85,B 0,C 180,E1 -20080.677,E2 -20080.677} C_VEL
LIN {X 0,Y 377.987,Z 570.582,A -85,B 0,C 180,E1 -20082.845,E2 -20082.845} C_VEL
LIN {X 0,Y 378.261,Z 570.569,A -85,B 0,C 180,E1 -20085.022,E2 -20085.022} C_VEL
LIN {X 0,Y 378.712,Z 569.19,A -85,B 0,C 180,E1 -20087.21,E2 -20087.21} C_VEL
LIN {X 0,Y 379.494,Z 566.393,A -85,B 0,C 180,E1 -20089.401,E2 -20089.401} C_VEL
LIN {X 0,Y 380.623,Z 562.083,A -85,B 0,C 180,E1 -20091.592,E2 -20091.592} C_VEL
LIN {X 0,Y 381.822,Z 557.046,A -85,B 0,C 180,E1 -20093.474,E2 -20093.474} C_VEL
LIN {X 0,Y 383.438,Z 550.352,A -85,B 0,C 180,E1 -20095.419,E2 -20095.419} C_VEL
LIN {X 0,Y 385.102,Z 543.358,A -85,B 0,C 180,E1 -20097.043,E2 -20097.043} C_VEL
LIN {X 0,Y 386.922,Z 534.896,A -85,B 0,C 180,E1 -20098.664,E2 -20098.664} C_VEL
LIN {X 0,Y 389.038,Z 524.623,A -85,B 0,C 180,E1 -20100.27,E2 -20100.27} C_VEL
LIN {X 0,Y 390.97,Z 514.185,A -85,B 0,C 180,E1 -20101.599,E2 -20101.599} C_VEL
LIN {X 0,Y 392.893,Z 502.585,A -85,B 0,C 180,E1 -20102.804,E2 -20102.804} C_VEL
LIN {X 0,Y 394.58,Z 490.204,A -85,B 0,C 180,E1 -20103.842,E2 -20103.842} C_VEL
LIN {X 0,Y 396.019,Z 477.23,A -85,B 0,C 180,E1 -20104.698,E2 -20104.698} C_VEL
LIN {X 0,Y 397.067,Z 464.876,A -85,B 0,C 180,E1 -20105.326,E2 -20105.326} C_VEL
LIN {X 0,Y 397.908,Z 451.233,A -85,B 0,C 180,E1 -20105.822,E2 -20105.822} C_VEL
LIN {X 0,Y 398.459,Z 433.178,A -85,B 0,C 180,E1 -20106.222,E2 -20106.222} C_VEL
LIN {X 0,Y 399.426,Z 400.229,A -85,B 0,C 180,E1 -20106.815,E2 -20106.815} C_VEL
LIN {X 0,Y 398.902,Z 394.43,A -85,B 0,C 180,E1 -20106.975,E2 -20106.975} C_VEL
LIN {X 0,Y 394.505,Z 375.787,A -85,B 0,C 180,E1 -20107.726,E2 -20107.726} C_VEL
LIN {X 0,Y 394.244,Z 369.983,A -85,B 0,C 180,E1 -20107.87,E2 -20107.87} C_VEL
LIN {X 0,Y 394.553,Z 355.805,A -85,B 0,C 180,E1 -20108.139,E2 -20108.139} C_VEL
LIN {X 0,Y 387.199,Z 339.264,A -85,B 0,C 180,E1 -20109.146,E2 -20109.146} C_VEL
LIN {X 0,Y 378.958,Z 322.986,A -85,B 0,C 180,E1 -20110.288,E2 -20110.288} C_VEL
LIN {X 0,Y 373.509,Z 312.804,A -85,B 0,C 180,E1 -20111.072,E2 -20111.072} C_VEL
LIN {X 0,Y 372.981,Z 310.573,A -85,B 0,C 180,E1 -20111.87,E2 -20111.87} C_VEL
LIN {X 0,Y 373.025,Z 310.562,A -85,B 0,C 180,E1 -20115.519,E2 -20115.519} C_VEL
LIN {X 0,Y 372.983,Z 310.583,A -85,B 0,C 180,E1 -20118.907,E2 -20118.907} C_VEL
LIN {X 0,Y 373.029,Z 310.575,A -85,B 0,C 180,E1 -20122.053,E2 -20122.053} C_VEL
LIN {X 0,Y 373.047,Z 310.555,A -85,B 0,C 180,E1 -20125.7,E2 -20125.7} C_VEL
LIN {X 0,Y 373.045,Z 310.567,A -85,B 0,C 180,E1 -20129.538,E2 -20129.538} C_VEL
LIN {X 0,Y 373.064,Z 310.562,A -85,B 0,C 180,E1 -20133.217,E2 -20133.217} C_VEL
LIN {X 0,Y 373.067,Z 310.559,A -85,B 0,C 180,E1 -20136.915,E2 -20136.915} C_VEL
LIN {X 0,Y 373.12,Z 310.557,A -85,B 0,C 180,E1 -20140.251,E2 -20140.251} C_VEL
LIN {X 0,Y 373.11,Z 310.567,A -85,B 0,C 180,E1 -20143.644,E2 -20143.644} C_VEL
LIN {X 0,Y 373.21,Z 310.548,A -85,B 0,C 180,E1 -20147.39,E2 -20147.39} C_VEL
LIN {X 0,Y 373.279,Z 310.53,A -85,B 0,C 180,E1 -20151.366,E2 -20151.366} C_VEL
LIN {X 0,Y 373.362,Z 310.534,A -85,B 0,C 180,E1 -20154.618,E2 -20154.618} C_VEL
LIN {X 0,Y 373.386,Z 310.514,A -85,B 0,C 180,E1 -20156.774,E2 -20156.774} C_VEL
LIN {X 0,Y 373.364,Z 310.531,A -85,B 0,C 180,E1 -20160,E2 -20160} C_VEL
LIN {X 0,Y 373.389,Z 310.522,A -85,B 0,C 180,E1 -20163.226,E2 -20163.226} C_VEL
LIN {X 0,Y 373.356,Z 310.523,A -85,B 0,C 180,E1 -20166.463,E2 -20166.463} C_VEL
LIN {X 0,Y 373.243,Z 310.546,A -85,B 0,C 180,E1 -20169.724,E2 -20169.724} C_VEL
LIN {X 0,Y 373.22,Z 310.535,A -85,B 0,C 180,E1 -20173.015,E2 -20173.015} C_VEL
LIN {X 0,Y 373.158,Z 310.545,A -85,B 0,C 180,E1 -20176.815,E2 -20176.815} C_VEL
LIN {X 0,Y 373.121,Z 310.563,A -85,B 0,C 180,E1 -20180.188,E2 -20180.188} C_VEL
LIN {X 0,Y 373.059,Z 310.566,A -85,B 0,C 180,E1 -20183.222,E2 -20183.222} C_VEL
LIN {X 0,Y 373.064,Z 310.562,A -85,B 0,C 180,E1 -20186.783,E2 -20186.783} C_VEL
LIN {X 0,Y 373.055,Z 310.564,A -85,B 0,C 180,E1 -20190.461,E2 -20190.461} C_VEL
LIN {X 0,Y 373.07,Z 310.547,A -85,B 0,C 180,E1 -20194.281,E2 -20194.281} C_VEL
LIN {X 0,Y 373.094,Z 310.54,A -85,B 0,C 180,E1 -20196.925,E2 -20196.925} C_VEL
LIN {X 0,Y 373.065,Z 310.569,A -85,B 0,C 180,E1 -20199.67,E2 -20199.67} C_VEL
LIN {X 0,Y 373.081,Z 310.571,A -85,B 0,C 180,E1 -20204,E2 -20204} C_VEL
LIN {X 0,Y 373.04,Z 310.572,A -85,B 0,C 180,E1 -20207.476,E2 -20207.476} C_VEL
LIN {X 0,Y 373.068,Z 310.575,A -85,B 0,C 180,E1 -20210.335,E2 -20210.335} C_VEL
LIN {X 0,Y 373.097,Z 310.758,A -85,B 0,C 180,E1 -20211.88,E2 -20211.88} C_VEL
LIN {X 0,Y 375.874,Z 320.784,A -85,B 0,C 180,E1 -20214.716,E2 -20214.716} C_VEL
LIN {X 0,Y 378.517,Z 331.536,A -85,B 0,C 180,E1 -20217.548,E2 -20217.548} C_VEL
LIN {X 0,Y 381.362,Z 345.004,A -85,B 0,C 180,E1 -20220.878,E2 -20220.878} C_VEL
LIN {X 0,Y 382.16,Z 349.299,A -85,B 0,C 180,E1 -20221.85,E2 -20221.85} C_VEL
LIN {X 0,Y 384.048,Z 356.77,A -85,B 0,C 180,E1 -20222.19,E2 -20222.19} C_VEL
LIN {X 0,Y 389.897,Z 388.164,A -85,B 0,C 180,E1 -20223.384,E2 -20223.384} C_VEL
LIN {X 0,Y 393.058,Z 409.79,A -85,B 0,C 180,E1 -20224.106,E2 -20224.106} C_VEL
LIN {X 0,Y 390.788,Z 487.302,A -85,B 0,C 180,E1 -20225.551,E2 -20225.551} C_VEL
LIN {X 0,Y 389.75,Z 501.982,A -85,B 0,C 180,E1 -20226.011,E2 -20226.011} C_VEL
LIN {X 0,Y 388.198,Z 515.417,A -85,B 0,C 180,E1 -20226.615,E2 -20226.615} C_VEL
LIN {X 0,Y 386.487,Z 527.669,A -85,B 0,C 180,E1 -20227.352,E2 -20227.352} C_VEL
LIN {X 0,Y 384.413,Z 540.556,A -85,B 0,C 180,E1 -20228.353,E2 -20228.353} C_VEL
LIN {X 0,Y 382.137,Z 553.386,A -85,B 0,C 180,E1 -20229.622,E2 -20229.622} C_VEL
LIN {X 0,Y 379.969,Z 563.927,A -85,B 0,C 180,E1 -20230.904,E2 -20230.904} C_VEL
LIN {X 0,Y 377.677,Z 574.423,A -85,B 0,C 180,E1 -20232.463,E2 -20232.463} C_VEL
LIN {X 0,Y 375.775,Z 583.12,A -85,B 0,C 180,E1 -20234.045,E2 -20234.045} C_VEL
LIN {X 0,Y 374.065,Z 591.507,A -85,B 0,C 180,E1 -20235.914,E2 -20235.914} C_VEL
LIN {X 0,Y 372.712,Z 598.156,A -85,B 0,C 180,E1 -20237.754,E2 -20237.754} C_VEL
LIN {X 0,Y 371.649,Z 603.719,A -85,B 0,C 180,E1 -20239.689,E2 -20239.689} C_VEL
LIN {X 0,Y 371.077,Z 607.378,A -85,B 0,C 180,E1 -20241.317,E2 -20241.317} C_VEL
LIN {X 0,Y 370.743,Z 611.012,A -85,B 0,C 180,E1 -20243.494,E2 -20243.494} C_VEL
LIN {X 0,Y 370.741,Z 613.112,A -85,B 0,C 180,E1 -20245.126,E2 -20245.126} C_VEL
LIN {X 0,Y 370.697,Z 617.042,A -85,B 0,C 180,E1 -20246.753,E2 -20246.753} C_VEL
LIN {X 0,Y 370.742,Z 620.788,A -85,B 0,C 180,E1 -20248.92,E2 -20248.92} C_VEL
LIN {X 0,Y 370.655,Z 622.989,A -85,B 0,C 180,E1 -20251.085,E2 -20251.085} C_VEL
LIN {X 0,Y 370.548,Z 623.725,A -85,B 0,C 180,E1 -20253.254,E2 -20253.254} C_VEL
LIN {X 0,Y 370.721,Z 623.027,A -85,B 0,C 180,E1 -20255.423,E2 -20255.423} C_VEL
LIN {X 0,Y 371.078,Z 620.89,A -85,B 0,C 180,E1 -20257.595,E2 -20257.595} C_VEL
LIN {X 0,Y 371.929,Z 617.289,A -85,B 0,C 180,E1 -20259.761,E2 -20259.761} C_VEL
LIN {X 0,Y 373.354,Z 612.142,A -85,B 0,C 180,E1 -20261.912,E2 -20261.912} C_VEL
LIN {X 0,Y 374.717,Z 606.496,A -85,B 0,C 180,E1 -20263.728,E2 -20263.728} C_VEL
LIN {X 0,Y 376.752,Z 598.974,A -85,B 0,C 180,E1 -20265.642,E2 -20265.642} C_VEL
LIN {X 0,Y 379.132,Z 589.999,A -85,B 0,C 180,E1 -20267.473,E2 -20267.473} C_VEL
LIN {X 0,Y 381.392,Z 580.698,A -85,B 0,C 180,E1 -20269.028,E2 -20269.028} C_VEL
LIN {X 0,Y 384.15,Z 569.422,A -85,B 0,C 180,E1 -20270.551,E2 -20270.551} C_VEL
LIN {X 0,Y 386.591,Z 558.201,A -85,B 0,C 180,E1 -20271.806,E2 -20271.806} C_VEL
LIN {X 0,Y 389.373,Z 544.506,A -85,B 0,C 180,E1 -20273.035,E2 -20273.035} C_VEL
LIN {X 0,Y 391.737,Z 530.882,A -85,B 0,C 180,E1 -20274.005,E2 -20274.005} C_VEL
LIN {X 0,Y 394.034,Z 515.798,A -85,B 0,C 180,E1 -20274.811,E2 -20274.811} C_VEL
LIN {X 0,Y 395.906,Z 500.27,A -85,B 0,C 180,E1 -20275.408,E2 -20275.408} C_VEL
LIN {X 0,Y 402.762,Z 412.267,A -85,B 0,C 180,E1 -20277.872,E2 -20277.872} C_VEL
LIN {X 0,Y 401.714,Z 393.567,A -85,B 0,C 180,E1 -20278.779,E2 -20278.779} C_VEL
LIN {X 0,Y 400.116,Z 378.076,A -85,B 0,C 180,E1 -20279.676,E2 -20279.676} C_VEL
LIN {X 0,Y 397.958,Z 362.28,A -85,B 0,C 180,E1 -20280.728,E2 -20280.728} C_VEL
LIN {X 0,Y 394.699,Z 352.477,A -85,B 0,C 180,E1 -20281.811,E2 -20281.811} C_VEL
LIN {X 0,Y 393.662,Z 347.608,A -85,B 0,C 180,E1 -20282.616,E2 -20282.616} C_VEL
LIN {X 0,Y 390.125,Z 340.689,A -85,B 0,C 180,E1 -20284.32,E2 -20284.32} C_VEL
LIN {X 0,Y 386.563,Z 334.149,A -85,B 0,C 180,E1 -20286.274,E2 -20286.274} C_VEL
LIN {X 0,Y 383.239,Z 328.433,A -85,B 0,C 180,E1 -20288.422,E2 -20288.422} C_VEL
LIN {X 0,Y 381.201,Z 324.906,A -85,B 0,C 180,E1 -20290.027,E2 -20290.027} C_VEL
LIN {X 0,Y 379.379,Z 322.13,A -85,B 0,C 180,E1 -20291.659,E2 -20291.659} C_VEL
LIN {X 0,Y 378.961,Z 320.836,A -85,B 0,C 180,E1 -20292.325,E2 -20292.325} C_VEL
LIN {X 0,Y 376.802,Z 318.041,A -85,B 0,C 180,E1 -20295.058,E2 -20295.058} C_VEL
LIN {X 0,Y 376.013,Z 316.053,A -85,B 0,C 180,E1 -20297.885,E2 -20297.885} C_VEL
LIN {X 0,Y 375.884,Z 315.68,A -85,B 0,C 180,E1 -20299.823,E2 -20299.823} C_VEL
LIN {X 0,Y 375.983,Z 316.301,A -85,B 0,C 180,E1 -20302.064,E2 -20302.064} C_VEL
LIN {X 0,Y 376.777,Z 318.223,A -85,B 0,C 180,E1 -20304.886,E2 -20304.886} C_VEL
LIN {X 0,Y 377.906,Z 319.651,A -85,B 0,C 180,E1 -20306.522,E2 -20306.522} C_VEL
LIN {X 0,Y 380.249,Z 325.231,A -85,B 0,C 180,E1 -20310.175,E2 -20310.175} C_VEL
LIN {X 0,Y 382.457,Z 330.455,A -85,B 0,C 180,E1 -20312.751,E2 -20312.751} C_VEL
LIN {X 0,Y 385.288,Z 337.909,A -85,B 0,C 180,E1 -20315.727,E2 -20315.727} C_VEL
LIN {X 0,Y 387.79,Z 345.987,A -85,B 0,C 180,E1 -20318.388,E2 -20318.388} C_VEL
LIN {X 0,Y 388.588,Z 348.572,A -85,B 0,C 180,E1 -20319.122,E2 -20319.122} C_VEL
LIN {X 0,Y 392.998,Z 356.399,A -85,B 0,C 180,E1 -20320.391,E2 -20320.391} C_VEL
LIN {X 0,Y 398.304,Z 366.714,A -85,B 0,C 180,E1 -20321.807,E2 -20321.807} C_VEL
LIN {X 0,Y 401.416,Z 374.153,A -85,B 0,C 180,E1 -20322.636,E2 -20322.636} C_VEL
LIN {X 0,Y 403.754,Z 388.518,A -85,B 0,C 180,E1 -20323.586,E2 -20323.586} C_VEL
LIN {X 0,Y 404.406,Z 394.322,A -85,B 0,C 180,E1 -20323.911,E2 -20323.911} C_VEL
LIN {X 0,Y 396.677,Z 489.811,A -85,B 0,C 180,E1 -20326.552,E2 -20326.552} C_VEL
LIN {X 0,Y 394.912,Z 505.315,A -85,B 0,C 180,E1 -20327.21,E2 -20327.21} C_VEL
LIN {X 0,Y 392.885,Z 519.703,A -85,B 0,C 180,E1 -20328.039,E2 -20328.039} C_VEL
LIN {X 0,Y 390.574,Z 532.964,A -85,B 0,C 180,E1 -20329.015,E2 -20329.015} C_VEL
LIN {X 0,Y 387.932,Z 546.23,A -85,B 0,C 180,E1 -20330.254,E2 -20330.254} C_VEL
LIN {X 0,Y 385.267,Z 558.208,A -85,B 0,C 180,E1 -20331.637,E2 -20331.637} C_VEL
LIN {X 0,Y 382.722,Z 568.943,A -85,B 0,C 180,E1 -20333.168,E2 -20333.168} C_VEL
LIN {X 0,Y 380.414,Z 577.884,A -85,B 0,C 180,E1 -20334.718,E2 -20334.718} C_VEL
LIN {X 0,Y 377.885,Z 586.514,A -85,B 0,C 180,E1 -20336.546,E2 -20336.546} C_VEL
LIN {X 0,Y 375.794,Z 593.509,A -85,B 0,C 180,E1 -20338.398,E2 -20338.398} C_VEL
LIN {X 0,Y 373.914,Z 599.759,A -85,B 0,C 180,E1 -20340.537,E2 -20340.537} C_VEL
LIN {X 0,Y 372.877,Z 603.32,A -85,B 0,C 180,E1 -20342.153,E2 -20342.153} C_VEL
LIN {X 0,Y 371.882,Z 606.758,A -85,B 0,C 180,E1 -20344.321,E2 -20344.321} C_VEL
LIN {X 0,Y 371.094,Z 608.768,A -85,B 0,C 180,E1 -20346.503,E2 -20346.503} C_VEL
LIN {X 0,Y 370.627,Z 609.324,A -85,B 0,C 180,E1 -20348.696,E2 -20348.696} C_VEL
LIN {X 0,Y 370.465,Z 608.679,A -85,B 0,C 180,E1 -20350.516,E2 -20350.516} C_VEL
LIN {X 0,Y 370.337,Z 607.382,A -85,B 0,C 180,E1 -20352.008,E2 -20352.008} C_VEL
LIN {X 0,Y 370.389,Z 604.187,A -85,B 0,C 180,E1 -20354.232,E2 -20354.232} C_VEL
LIN {X 0,Y 370.541,Z 600.832,A -85,B 0,C 180,E1 -20355.852,E2 -20355.852} C_VEL
LIN {X 0,Y 370.713,Z 596.177,A -85,B 0,C 180,E1 -20357.597,E2 -20357.597} C_VEL
LIN {X 0,Y 371.025,Z 589.868,A -85,B 0,C 180,E1 -20359.459,E2 -20359.459} C_VEL
LIN {X 0,Y 371.509,Z 582.184,A -85,B 0,C 180,E1 -20361.281,E2 -20361.281} C_VEL
LIN {X 0,Y 372.13,Z 572.777,A -85,B 0,C 180,E1 -20363.097,E2 -20363.097} C_VEL
LIN {X 0,Y 372.912,Z 562.64,A -85,B 0,C 180,E1 -20364.704,E2 -20364.704} C_VEL
LIN {X 0,Y 373.719,Z 551.571,A -85,B 0,C 180,E1 -20366.148,E2 -20366.148} C_VEL
LIN {X 0,Y 374.725,Z 538.345,A -85,B 0,C 180,E1 -20367.557,E2 -20367.557} C_VEL
LIN {X 0,Y 375.63,Z 525.46,A -85,B 0,C 180,E1 -20368.668,E2 -20368.668} C_VEL
LIN {X 0,Y 376.474,Z 511.53,A -85,B 0,C 180,E1 -20369.617,E2 -20369.617} C_VEL
LIN {X 0,Y 377.291,Z 496.462,A -85,B 0,C 180,E1 -20370.391,E2 -20370.391} C_VEL
LIN {X 0,Y 377.966,Z 480.977,A -85,B 0,C 180,E1 -20370.948,E2 -20370.948} C_VEL
LIN {X 0,Y 380.893,Z 380.443,A -85,B 0,C 180,E1 -20373.508,E2 -20373.508} C_VEL
LIN {X 0,Y 376.952,Z 346.634,A -85,B 0,C 180,E1 -20374.545,E2 -20374.545} C_VEL
LIN {X 0,Y 376.86,Z 345.045,A -85,B 0,C 180,E1 -20374.616,E2 -20374.616} C_VEL
LIN {X 0,Y 377.592,Z 333.082,A -85,B 0,C 180,E1 -20376.615,E2 -20376.615} C_VEL
LIN {X 0,Y 374.011,Z 315.092,A -85,B 0,C 180,E1 -20379.836,E2 -20379.836} C_VEL
LIN {X 0,Y 373.025,Z 310.579,A -85,B 0,C 180,E1 -20380.664,E2 -20380.664} C_VEL
LIN {X 0,Y 373.047,Z 310.573,A -85,B 0,C 180,E1 -20384.477,E2 -20384.477} C_VEL
LIN {X 0,Y 372.974,Z 310.58,A -85,B 0,C 180,E1 -20387.459,E2 -20387.459} C_VEL
LIN {X 0,Y 373.02,Z 310.578,A -85,B 0,C 180,E1 -20390.344,E2 -20390.344} C_VEL
LIN {X 0,Y 373.045,Z 310.574,A -85,B 0,C 180,E1 -20393.841,E2 -20393.841} C_VEL
LIN {X 0,Y 372.996,Z 310.574,A -85,B 0,C 180,E1 -20397.001,E2 -20397.001} C_VEL
LIN {X 0,Y 373.026,Z 310.572,A -85,B 0,C 180,E1 -20400.774,E2 -20400.774} C_VEL
LIN {X 0,Y 373.081,Z 310.57,A -85,B 0,C 180,E1 -20404.415,E2 -20404.415} C_VEL
LIN {X 0,Y 373.076,Z 310.573,A -85,B 0,C 180,E1 -20407.943,E2 -20407.943} C_VEL
LIN {X 0,Y 373.148,Z 310.562,A -85,B 0,C 180,E1 -20410.25,E2 -20410.25} C_VEL
LIN {X 0,Y 373.198,Z 310.554,A -85,B 0,C 180,E1 -20413.646,E2 -20413.646} C_VEL
LIN {X 0,Y 373.271,Z 310.548,A -85,B 0,C 180,E1 -20417.96,E2 -20417.96} C_VEL
LIN {X 0,Y 373.318,Z 310.893,A -85,B 0,C 180,E1 -20418.171,E2 -20418.171} C_VEL
LIN {X 0,Y 382.237,Z 336.793,A -85,B 0,C 180,E1 -20419.173,E2 -20419.173} C_VEL
LIN {X 0,Y 383.766,Z 341.691,A -85,B 0,C 180,E1 -20419.348,E2 -20419.348} C_VEL
LIN {X 0,Y 381.449,Z 446.934,A -85,B 0,C 180,E1 -20421.317,E2 -20421.317} C_VEL
LIN {X 0,Y 380.907,Z 461.246,A -85,B 0,C 180,E1 -20421.804,E2 -20421.804} C_VEL
LIN {X 0,Y 380.162,Z 475.559,A -85,B 0,C 180,E1 -20422.521,E2 -20422.521} C_VEL
LIN {X 0,Y 379.171,Z 488.312,A -85,B 0,C 180,E1 -20423.368,E2 -20423.368} C_VEL
LIN {X 0,Y 378.205,Z 499.303,A -85,B 0,C 180,E1 -20424.284,E2 -20424.284} C_VEL
LIN {X 0,Y 376.854,Z 510.943,A -85,B 0,C 180,E1 -20425.467,E2 -20425.467} C_VEL
LIN {X 0,Y 375.881,Z 521.523,A -85,B 0,C 180,E1 -20426.793,E2 -20426.793} C_VEL
LIN {X 0,Y 374.803,Z 530.45,A -85,B 0,C 180,E1 -20428.123,E2 -20428.123} C_VEL
LIN {X 0,Y 373.707,Z 539.431,A -85,B 0,C 180,E1 -20429.729,E2 -20429.729} C_VEL
LIN {X 0,Y 372.799,Z 546.917,A -85,B 0,C 180,E1 -20431.343,E2 -20431.343} C_VEL
LIN {X 0,Y 372.218,Z 554.042,A -85,B 0,C 180,E1 -20433.234,E2 -20433.234} C_VEL
LIN {X 0,Y 371.775,Z 559.049,A -85,B 0,C 180,E1 -20434.861,E2 -20434.861} C_VEL
LIN {X 0,Y 371.225,Z 564.233,A -85,B 0,C 180,E1 -20437.042,E2 -20437.042} C_VEL
LIN {X 0,Y 370.976,Z 567.159,A -85,B 0,C 180,E1 -20438.685,E2 -20438.685} C_VEL
LIN {X 0,Y 370.902,Z 569.775,A -85,B 0,C 180,E1 -20440.883,E2 -20440.883} C_VEL
LIN {X 0,Y 370.927,Z 571.026,A -85,B 0,C 180,E1 -20443.094,E2 -20443.094} C_VEL
LIN {X 0,Y 371.24,Z 570.921,A -85,B 0,C 180,E1 -20445.313,E2 -20445.313} C_VEL
LIN {X 0,Y 371.734,Z 569.451,A -85,B 0,C 180,E1 -20447.544,E2 -20447.544} C_VEL
LIN {X 0,Y 372.587,Z 566.56,A -85,B 0,C 180,E1 -20449.776,E2 -20449.776} C_VEL
LIN {X 0,Y 373.792,Z 562.151,A -85,B 0,C 180,E1 -20452.007,E2 -20452.007} C_VEL
LIN {X 0,Y 374.955,Z 557.531,A -85,B 0,C 180,E1 -20453.744,E2 -20453.744} C_VEL
LIN {X 0,Y 376.531,Z 551.227,A -85,B 0,C 180,E1 -20455.624,E2 -20455.624} C_VEL
LIN {X 0,Y 378.248,Z 544.371,A -85,B 0,C 180,E1 -20457.268,E2 -20457.268} C_VEL
LIN {X 0,Y 380.132,Z 535.998,A -85,B 0,C 180,E1 -20458.923,E2 -20458.923} C_VEL
LIN {X 0,Y 382.311,Z 525.836,A -85,B 0,C 180,E1 -20460.559,E2 -20460.559} C_VEL
LIN {X 0,Y 384.494,Z 514.488,A -85,B 0,C 180,E1 -20462.041,E2 -20462.041} C_VEL
LIN {X 0,Y 386.608,Z 502.254,A -85,B 0,C 180,E1 -20463.315,E2 -20463.315} C_VEL
LIN {X 0,Y 388.255,Z 490.445,A -85,B 0,C 180,E1 -20464.314,E2 -20464.314} C_VEL
LIN {X 0,Y 389.723,Z 477.413,A -85,B 0,C 180,E1 -20465.184,E2 -20465.184} C_VEL
LIN {X 0,Y 390.881,Z 464.195,A -85,B 0,C 180,E1 -20465.852,E2 -20465.852} C_VEL
LIN {X 0,Y 391.734,Z 450.544,A -85,B 0,C 180,E1 -20466.339,E2 -20466.339} C_VEL
LIN {X 0,Y 392.308,Z 430.489,A -85,B 0,C 180,E1 -20466.773,E2 -20466.773} C_VEL
LIN {X 0,Y 394.244,Z 369.983,A -85,B 0,C 180,E1 -20467.87,E2 -20467.87} C_VEL
LIN {X 0,Y 393.804,Z 366.201,A -85,B 0,C 180,E1 -20467.986,E2 -20467.986} C_VEL
LIN {X 0,Y 392.415,Z 362.736,A -85,B 0,C 180,E1 -20468.179,E2 -20468.179} C_VEL
LIN {X 0,Y 386.46,Z 353.094,A -85,B 0,C 180,E1 -20468.916,E2 -20468.916} C_VEL
LIN {X 0,Y 385.927,Z 351.917,A -85,B 0,C 180,E1 -20468.99,E2 -20468.99} C_VEL
LIN {X 0,Y 376.773,Z 332.603,A -85,B 0,C 180,E1 -20470.289,E2 -20470.289} C_VEL
LIN {X 0,Y 368.002,Z 316.467,A -85,B 0,C 180,E1 -20471.56,E2 -20471.56} C_VEL
LIN {X 0,Y 366.405,Z 313.239,A -85,B 0,C 180,E1 -20471.827,E2 -20471.827} C_VEL
LIN {X 0,Y 365.941,Z 311.455,A -85,B 0,C 180,E1 -20472.506,E2 -20472.506} C_VEL
LIN {X 0,Y 365.98,Z 311.438,A -85,B 0,C 180,E1 -20475.079,E2 -20475.079} C_VEL
LIN {X 0,Y 365.947,Z 311.457,A -85,B 0,C 180,E1 -20478.282,E2 -20478.282} C_VEL
LIN {X 0,Y 365.976,Z 311.451,A -85,B 0,C 180,E1 -20482.233,E2 -20482.233} C_VEL
LIN {X 0,Y 365.996,Z 311.427,A -85,B 0,C 180,E1 -20485.374,E2 -20485.374} C_VEL
LIN {X 0,Y 365.97,Z 311.447,A -85,B 0,C 180,E1 -20488.885,E2 -20488.885} C_VEL
LIN {X 0,Y 366.002,Z 311.44,A -85,B 0,C 180,E1 -20492.658,E2 -20492.658} C_VEL
LIN {X 0,Y 366.002,Z 311.44,A -85,B 0,C 180,E1 -20496.303,E2 -20496.303} C_VEL
LIN {X 0,Y 366.091,Z 311.435,A -85,B 0,C 180,E1 -20499.855,E2 -20499.855} C_VEL
LIN {X 0,Y 366.075,Z 311.444,A -85,B 0,C 180,E1 -20503.321,E2 -20503.321} C_VEL
LIN {X 0,Y 366.177,Z 311.423,A -85,B 0,C 180,E1 -20507.29,E2 -20507.29} C_VEL
LIN {X 0,Y 366.214,Z 311.409,A -85,B 0,C 180,E1 -20511.198,E2 -20511.198} C_VEL
LIN {X 0,Y 366.318,Z 311.411,A -85,B 0,C 180,E1 -20514.514,E2 -20514.514} C_VEL
LIN {X 0,Y 366.346,Z 311.39,A -85,B 0,C 180,E1 -20516.712,E2 -20516.712} C_VEL
LIN {X 0,Y 366.329,Z 311.408,A -85,B 0,C 180,E1 -20520,E2 -20520} C_VEL
LIN {X 0,Y 366.349,Z 311.399,A -85,B 0,C 180,E1 -20523.288,E2 -20523.288} C_VEL
LIN {X 0,Y 366.355,Z 311.398,A -85,B 0,C 180,E1 -20526.206,E2 -20526.206} C_VEL
LIN {X 0,Y 366.204,Z 311.422,A -85,B 0,C 180,E1 -20529.913,E2 -20529.913} C_VEL
LIN {X 0,Y 366.168,Z 311.415,A -85,B 0,C 180,E1 -20533.271,E2 -20533.271} C_VEL
LIN {X 0,Y 366.103,Z 311.422,A -85,B 0,C 180,E1 -20536.95,E2 -20536.95} C_VEL
LIN {X 0,Y 366.057,Z 311.444,A -85,B 0,C 180,E1 -20540.357,E2 -20540.357} C_VEL
LIN {X 0,Y 366.002,Z 311.448,A -85,B 0,C 180,E1 -20543.697,E2 -20543.697} C_VEL
LIN {X 0,Y 366.002,Z 311.446,A -85,B 0,C 180,E1 -20547.342,E2 -20547.342} C_VEL
LIN {X 0,Y 365.984,Z 311.448,A -85,B 0,C 180,E1 -20551.114,E2 -20551.114} C_VEL
LIN {X 0,Y 366.006,Z 311.421,A -85,B 0,C 180,E1 -20554.629,E2 -20554.629} C_VEL
LIN {X 0,Y 366.065,Z 311.433,A -85,B 0,C 180,E1 -20557.756,E2 -20557.756} C_VEL
LIN {X 0,Y 365.986,Z 311.449,A -85,B 0,C 180,E1 -20560.595,E2 -20560.595} C_VEL
LIN {X 0,Y 366.029,Z 311.447,A -85,B 0,C 180,E1 -20563.544,E2 -20563.544} C_VEL
LIN {X 0,Y 366.029,Z 311.448,A -85,B 0,C 180,E1 -20566.651,E2 -20566.651} C_VEL
LIN {X 0,Y 366.012,Z 311.451,A -85,B 0,C 180,E1 -20569.951,E2 -20569.951} C_VEL
LIN {X 0,Y 366.035,Z 311.57,A -85,B 0,C 180,E1 -20571.195,E2 -20571.195} C_VEL
LIN {X 0,Y 368.659,Z 320.883,A -85,B 0,C 180,E1 -20573.918,E2 -20573.918} C_VEL
LIN {X 0,Y 371.625,Z 332.793,A -85,B 0,C 180,E1 -20577.167,E2 -20577.167} C_VEL
LIN {X 0,Y 374.489,Z 346.385,A -85,B 0,C 180,E1 -20580.599,E2 -20580.599} C_VEL
LIN {X 0,Y 374.937,Z 348.669,A -85,B 0,C 180,E1 -20581.139,E2 -20581.139} C_VEL
LIN {X 0,Y 377.314,Z 354.893,A -85,B 0,C 180,E1 -20581.511,E2 -20581.511} C_VEL
LIN {X 0,Y 383.144,Z 385.499,A -85,B 0,C 180,E1 -20582.73,E2 -20582.73} C_VEL
LIN {X 0,Y 386.843,Z 410.396,A -85,B 0,C 180,E1 -20583.591,E2 -20583.591} C_VEL
LIN {X 0,Y 385.201,Z 467.943,A -85,B 0,C 180,E1 -20584.67,E2 -20584.67} C_VEL
LIN {X 0,Y 384.408,Z 489.653,A -85,B 0,C 180,E1 -20585.118,E2 -20585.118} C_VEL
LIN {X 0,Y 383.222,Z 504.147,A -85,B 0,C 180,E1 -20585.612,E2 -20585.612} C_VEL
LIN {X 0,Y 381.552,Z 517.478,A -85,B 0,C 180,E1 -20586.255,E2 -20586.255} C_VEL
LIN {X 0,Y 379.723,Z 530.063,A -85,B 0,C 180,E1 -20587.069,E2 -20587.069} C_VEL
LIN {X 0,Y 377.596,Z 542.445,A -85,B 0,C 180,E1 -20588.089,E2 -20588.089} C_VEL
LIN {X 0,Y 375.243,Z 554.841,A -85,B 0,C 180,E1 -20589.373,E2 -20589.373} C_VEL
LIN {X 0,Y 372.849,Z 565.996,A -85,B 0,C 180,E1 -20590.81,E2 -20590.81} C_VEL
LIN {X 0,Y 370.51,Z 576.032,A -85,B 0,C 180,E1 -20592.397,E2 -20592.397} C_VEL
LIN {X 0,Y 368.655,Z 584.401,A -85,B 0,C 180,E1 -20594.011,E2 -20594.011} C_VEL
LIN {X 0,Y 366.925,Z 592.44,A -85,B 0,C 180,E1 -20595.916,E2 -20595.916} C_VEL
LIN {X 0,Y 365.524,Z 598.955,A -85,B 0,C 180,E1 -20597.834,E2 -20597.834} C_VEL
LIN {X 0,Y 364.396,Z 604.782,A -85,B 0,C 180,E1 -20600.041,E2 -20600.041} C_VEL
LIN {X 0,Y 363.72,Z 609.079,A -85,B 0,C 180,E1 -20602.256,E2 -20602.256} C_VEL
LIN {X 0,Y 363.641,Z 611.972,A -85,B 0,C 180,E1 -20604.476,E2 -20604.476} C_VEL
LIN {X 0,Y 363.675,Z 612.736,A -85,B 0,C 180,E1 -20605.169,E2 -20605.169} C_VEL
LIN {X 0,Y 363.628,Z 617.538,A -85,B 0,C 180,E1 -20607.242,E2 -20607.242} C_VEL
LIN {X 0,Y 363.66,Z 620.328,A -85,B 0,C 180,E1 -20608.899,E2 -20608.899} C_VEL
LIN {X 0,Y 363.569,Z 622.664,A -85,B 0,C 180,E1 -20611.107,E2 -20611.107} C_VEL
LIN {X 0,Y 363.47,Z 623.532,A -85,B 0,C 180,E1 -20613.317,E2 -20613.317} C_VEL
LIN {X 0,Y 363.647,Z 622.972,A -85,B 0,C 180,E1 -20615.529,E2 -20615.529} C_VEL
LIN {X 0,Y 364.015,Z 621.006,A -85,B 0,C 180,E1 -20617.744,E2 -20617.744} C_VEL
LIN {X 0,Y 364.931,Z 617.592,A -85,B 0,C 180,E1 -20619.95,E2 -20619.95} C_VEL
LIN {X 0,Y 366.412,Z 612.62,A -85,B 0,C 180,E1 -20622.141,E2 -20622.141} C_VEL
LIN {X 0,Y 367.67,Z 607.856,A -85,B 0,C 180,E1 -20623.779,E2 -20623.779} C_VEL
LIN {X 0,Y 369.701,Z 600.96,A -85,B 0,C 180,E1 -20625.666,E2 -20625.666} C_VEL
LIN {X 0,Y 371.786,Z 593.784,A -85,B 0,C 180,E1 -20627.264,E2 -20627.264} C_VEL
LIN {X 0,Y 374.345,Z 583.677,A -85,B 0,C 180,E1 -20629.116,E2 -20629.116} C_VEL
LIN {X 0,Y 377.138,Z 573.134,A -85,B 0,C 180,E1 -20630.666,E2 -20630.666} C_VEL
LIN {X 0,Y 379.872,Z 561.55,A -85,B 0,C 180,E1 -20632.07,E2 -20632.07} C_VEL
LIN {X 0,Y 382.751,Z 548.737,A -85,B 0,C 180,E1 -20633.315,E2 -20633.315} C_VEL
LIN {X 0,Y 385.15,Z 536.159,A -85,B 0,C 180,E1 -20634.299,E2 -20634.299} C_VEL
LIN {X 0,Y 387.472,Z 522.92,A -85,B 0,C 180,E1 -20635.109,E2 -20635.109} C_VEL
LIN {X 0,Y 389.639,Z 507.769,A -85,B 0,C 180,E1 -20635.811,E2 -20635.811} C_VEL
LIN {X 0,Y 391.229,Z 491.656,A -85,B 0,C 180,E1 -20636.338,E2 -20636.338} C_VEL
LIN {X 0,Y 397.643,Z 412.833,A -85,B 0,C 180,E1 -20638.585,E2 -20638.585} C_VEL
LIN {X 0,Y 396.703,Z 394.959,A -85,B 0,C 180,E1 -20639.488,E2 -20639.488} C_VEL
LIN {X 0,Y 395.449,Z 381.483,A -85,B 0,C 180,E1 -20640.288,E2 -20640.288} C_VEL
LIN {X 0,Y 393.844,Z 368.341,A -85,B 0,C 180,E1 -20641.169,E2 -20641.169} C_VEL
LIN {X 0,Y 393.143,Z 364.535,A -85,B 0,C 180,E1 -20641.474,E2 -20641.474} C_VEL
LIN {X 0,Y 389.086,Z 352.975,A -85,B 0,C 180,E1 -20642.835,E2 -20642.835} C_VEL
LIN {X 0,Y 386.389,Z 347.327,A -85,B 0,C 180,E1 -20644.194,E2 -20644.194} C_VEL
LIN {X 0,Y 383.435,Z 341.814,A -85,B 0,C 180,E1 -20645.775,E2 -20645.775} C_VEL
LIN {X 0,Y 380.396,Z 336.363,A -85,B 0,C 180,E1 -20647.648,E2 -20647.648} C_VEL
LIN {X 0,Y 377.855,Z 331.928,A -85,B 0,C 180,E1 -20649.506,E2 -20649.506} C_VEL
LIN {X 0,Y 374.998,Z 326.961,A -85,B 0,C 180,E1 -20652.258,E2 -20652.258} C_VEL
LIN {X 0,Y 373.548,Z 324.959,A -85,B 0,C 180,E1 -20653.934,E2 -20653.934} C_VEL
LIN {X 0,Y 371.922,Z 322.155,A -85,B 0,C 180,E1 -20657.313,E2 -20657.313} C_VEL
LIN {X 0,Y 371.749,Z 321.441,A -85,B 0,C 180,E1 -20658.913,E2 -20658.913} C_VEL
LIN {X 0,Y 371.636,Z 321.69,A -85,B 0,C 180,E1 -20661.54,E2 -20661.54} C_VEL
LIN {X 0,Y 372.843,Z 324.465,A -85,B 0,C 180,E1 -20665.755,E2 -20665.755} C_VEL
LIN {X 0,Y 374.259,Z 327.804,A -85,B 0,C 180,E1 -20668.397,E2 -20668.397} C_VEL
LIN {X 0,Y 376.234,Z 332.181,A -85,B 0,C 180,E1 -20671.05,E2 -20671.05} C_VEL
LIN {X 0,Y 378.3,Z 337.691,A -85,B 0,C 180,E1 -20673.617,E2 -20673.617} C_VEL
LIN {X 0,Y 380.522,Z 344.076,A -85,B 0,C 180,E1 -20676.111,E2 -20676.111} C_VEL
LIN {X 0,Y 381.969,Z 348.724,A -85,B 0,C 180,E1 -20677.66,E2 -20677.66} C_VEL
LIN {X 0,Y 386.614,Z 356.727,A -85,B 0,C 180,E1 -20679.14,E2 -20679.14} C_VEL
LIN {X 0,Y 390.452,Z 363.802,A -85,B 0,C 180,E1 -20680.266,E2 -20680.266} C_VEL
LIN {X 0,Y 394.807,Z 372.796,A -85,B 0,C 180,E1 -20681.487,E2 -20681.487} C_VEL
LIN {X 0,Y 396.819,Z 377.85,A -85,B 0,C 180,E1 -20682.052,E2 -20682.052} C_VEL
LIN {X 0,Y 398.907,Z 391.661,A -85,B 0,C 180,E1 -20682.984,E2 -20682.984} C_VEL
LIN {X 0,Y 399.31,Z 396.06,A -85,B 0,C 180,E1 -20683.229,E2 -20683.229} C_VEL
LIN {X 0,Y 391.295,Z 489.874,A -85,B 0,C 180,E1 -20685.877,E2 -20685.877} C_VEL
LIN {X 0,Y 389.593,Z 504.28,A -85,B 0,C 180,E1 -20686.483,E2 -20686.483} C_VEL
LIN {X 0,Y 387.327,Z 519.726,A -85,B 0,C 180,E1 -20687.377,E2 -20687.377} C_VEL
LIN {X 0,Y 384.704,Z 533.945,A -85,B 0,C 180,E1 -20688.447,E2 -20688.447} C_VEL
LIN {X 0,Y 381.96,Z 547.062,A -85,B 0,C 180,E1 -20689.7,E2 -20689.7} C_VEL
LIN {X 0,Y 379.38,Z 557.908,A -85,B 0,C 180,E1 -20690.971,E2 -20690.971} C_VEL
LIN {X 0,Y 376.701,Z 568.727,A -85,B 0,C 180,E1 -20692.521,E2 -20692.521} C_VEL
LIN {X 0,Y 374.222,Z 577.726,A -85,B 0,C 180,E1 -20694.091,E2 -20694.091} C_VEL
LIN {X 0,Y 371.578,Z 586.402,A -85,B 0,C 180,E1 -20695.946,E2 -20695.946} C_VEL
LIN {X 0,Y 369.311,Z 593.441,A -85,B 0,C 180,E1 -20697.826,E2 -20697.826} C_VEL
LIN {X 0,Y 367.266,Z 599.742,A -85,B 0,C 180,E1 -20700,E2 -20700} C_VEL
LIN {X 0,Y 365.796,Z 604.385,A -85,B 0,C 180,E1 -20702.195,E2 -20702.195} C_VEL
LIN {X 0,Y 364.751,Z 607.481,A -85,B 0,C 180,E1 -20704.405,E2 -20704.405} C_VEL
LIN {X 0,Y 363.952,Z 609.154,A -85,B 0,C 180,E1 -20706.631,E2 -20706.631} C_VEL
LIN {X 0,Y 363.505,Z 609.4,A -85,B 0,C 180,E1 -20708.868,E2 -20708.868} C_VEL
LIN {X 0,Y 363.361,Z 608.661,A -85,B 0,C 180,E1 -20710.534,E2 -20710.534} C_VEL
LIN {X 0,Y 363.231,Z 607.034,A -85,B 0,C 180,E1 -20712.247,E2 -20712.247} C_VEL
LIN {X 0,Y 363.216,Z 605.486,A -85,B 0,C 180,E1 -20713.38,E2 -20713.38} C_VEL
LIN {X 0,Y 363.405,Z 601.537,A -85,B 0,C 180,E1 -20715.473,E2 -20715.473} C_VEL
LIN {X 0,Y 363.612,Z 596.666,A -85,B 0,C 180,E1 -20717.373,E2 -20717.373} C_VEL
LIN {X 0,Y 363.938,Z 589.863,A -85,B 0,C 180,E1 -20719.422,E2 -20719.422} C_VEL
LIN {X 0,Y 364.354,Z 582.842,A -85,B 0,C 180,E1 -20721.128,E2 -20721.128} C_VEL
LIN {X 0,Y 364.997,Z 573.507,A -85,B 0,C 180,E1 -20722.986,E2 -20722.986} C_VEL
LIN {X 0,Y 365.743,Z 563.542,A -85,B 0,C 180,E1 -20724.616,E2 -20724.616} C_VEL
LIN {X 0,Y 366.563,Z 552.691,A -85,B 0,C 180,E1 -20726.087,E2 -20726.087} C_VEL
LIN {X 0,Y 367.561,Z 539.648,A -85,B 0,C 180,E1 -20727.524,E2 -20727.524} C_VEL
LIN {X 0,Y 368.515,Z 526.158,A -85,B 0,C 180,E1 -20728.725,E2 -20728.725} C_VEL
LIN {X 0,Y 369.35,Z 512.346,A -85,B 0,C 180,E1 -20729.699,E2 -20729.699} C_VEL
LIN {X 0,Y 370.213,Z 497.558,A -85,B 0,C 180,E1 -20730.484,E2 -20730.484} C_VEL
LIN {X 0,Y 370.892,Z 482.519,A -85,B 0,C 180,E1 -20731.051,E2 -20731.051} C_VEL
LIN {X 0,Y 373.933,Z 381.072,A -85,B 0,C 180,E1 -20733.717,E2 -20733.717} C_VEL
LIN {X 0,Y 370.064,Z 347.355,A -85,B 0,C 180,E1 -20734.775,E2 -20734.775} C_VEL
LIN {X 0,Y 369.935,Z 345.118,A -85,B 0,C 180,E1 -20734.873,E2 -20734.873} C_VEL
LIN {X 0,Y 370.586,Z 334.236,A -85,B 0,C 180,E1 -20736.708,E2 -20736.708} C_VEL
LIN {X 0,Y 366.748,Z 315.093,A -85,B 0,C 180,E1 -20740.183,E2 -20740.183} C_VEL
LIN {X 0,Y 365.978,Z 311.456,A -85,B 0,C 180,E1 -20740.896,E2 -20740.896} C_VEL
LIN {X 0,Y 365.999,Z 311.447,A -85,B 0,C 180,E1 -20744.917,E2 -20744.917} C_VEL
LIN {X 0,Y 365.935,Z 311.463,A -85,B 0,C 180,E1 -20748.289,E2 -20748.289} C_VEL
LIN {X 0,Y 365.969,Z 311.453,A -85,B 0,C 180,E1 -20751.695,E2 -20751.695} C_VEL
LIN {X 0,Y 365.957,Z 311.449,A -85,B 0,C 180,E1 -20754.954,E2 -20754.954} C_VEL
LIN {X 0,Y 365.959,Z 311.455,A -85,B 0,C 180,E1 -20758.881,E2 -20758.881} C_VEL
LIN {X 0,Y 366.015,Z 311.447,A -85,B 0,C 180,E1 -20762.656,E2 -20762.656} C_VEL
LIN {X 0,Y 366.003,Z 311.449,A -85,B 0,C 180,E1 -20765.098,E2 -20765.098} C_VEL
LIN {X 0,Y 366.038,Z 311.445,A -85,B 0,C 180,E1 -20768.677,E2 -20768.677} C_VEL
LIN {X 0,Y 366.064,Z 311.441,A -85,B 0,C 180,E1 -20771.015,E2 -20771.015} C_VEL
LIN {X 0,Y 366.121,Z 311.437,A -85,B 0,C 180,E1 -20774.462,E2 -20774.462} C_VEL
LIN {X 0,Y 366.239,Z 311.529,A -85,B 0,C 180,E1 -20777.786,E2 -20777.786} C_VEL
LIN {X 0,Y 375.365,Z 337.703,A -85,B 0,C 180,E1 -20778.828,E2 -20778.828} C_VEL
LIN {X 0,Y 377.049,Z 343.494,A -85,B 0,C 180,E1 -20779.033,E2 -20779.033} C_VEL
LIN {X 0,Y 374.695,Z 446.624,A -85,B 0,C 180,E1 -20780.99,E2 -20780.99} C_VEL
LIN {X 0,Y 374.136,Z 461.185,A -85,B 0,C 180,E1 -20781.485,E2 -20781.485} C_VEL
LIN {X 0,Y 373.406,Z 475.059,A -85,B 0,C 180,E1 -20782.181,E2 -20782.181} C_VEL
LIN {X 0,Y 372.314,Z 488.887,A -85,B 0,C 180,E1 -20783.109,E2 -20783.109} C_VEL
LIN {X 0,Y 371.3,Z 499.855,A -85,B 0,C 180,E1 -20784.042,E2 -20784.042} C_VEL
LIN {X 0,Y 369.925,Z 511.471,A -85,B 0,C 180,E1 -20785.246,E2 -20785.246} C_VEL
LIN {X 0,Y 369.005,Z 521.071,A -85,B 0,C 180,E1 -20786.461,E2 -20786.461} C_VEL
LIN {X 0,Y 367.927,Z 530.135,A -85,B 0,C 180,E1 -20787.815,E2 -20787.815} C_VEL
LIN {X 0,Y 366.759,Z 539.243,A -85,B 0,C 180,E1 -20789.45,E2 -20789.45} C_VEL
LIN {X 0,Y 365.847,Z 546.83,A -85,B 0,C 180,E1 -20791.094,E2 -20791.094} C_VEL
LIN {X 0,Y 365.253,Z 553.143,A -85,B 0,C 180,E1 -20792.745,E2 -20792.745} C_VEL
LIN {X 0,Y 364.836,Z 558.33,A -85,B 0,C 180,E1 -20794.402,E2 -20794.402} C_VEL
LIN {X 0,Y 364.235,Z 563.848,A -85,B 0,C 180,E1 -20796.623,E2 -20796.623} C_VEL
LIN {X 0,Y 363.87,Z 567.796,A -85,B 0,C 180,E1 -20798.856,E2 -20798.856} C_VEL
LIN {X 0,Y 363.82,Z 570.306,A -85,B 0,C 180,E1 -20801.097,E2 -20801.097} C_VEL
LIN {X 0,Y 363.87,Z 571.468,A -85,B 0,C 180,E1 -20803.353,E2 -20803.353} C_VEL
LIN {X 0,Y 364.235,Z 571.274,A -85,B 0,C 180,E1 -20805.615,E2 -20805.615} C_VEL
LIN {X 0,Y 364.765,Z 569.716,A -85,B 0,C 180,E1 -20807.89,E2 -20807.89} C_VEL
LIN {X 0,Y 365.695,Z 566.689,A -85,B 0,C 180,E1 -20810.193,E2 -20810.193} C_VEL
LIN {X 0,Y 366.973,Z 562.223,A -85,B 0,C 180,E1 -20812.438,E2 -20812.438} C_VEL
LIN {X 0,Y 368.271,Z 557.399,A -85,B 0,C 180,E1 -20814.239,E2 -20814.239} C_VEL
LIN {X 0,Y 369.903,Z 551.082,A -85,B 0,C 180,E1 -20816.117,E2 -20816.117} C_VEL
LIN {X 0,Y 372.015,Z 542.791,A -85,B 0,C 180,E1 -20818.077,E2 -20818.077} C_VEL
LIN {X 0,Y 374.077,Z 534.017,A -85,B 0,C 180,E1 -20819.746,E2 -20819.746} C_VEL
LIN {X 0,Y 376.074,Z 524.892,A -85,B 0,C 180,E1 -20821.179,E2 -20821.179} C_VEL
LIN {X 0,Y 378.286,Z 513.593,A -85,B 0,C 180,E1 -20822.631,E2 -20822.631} C_VEL
LIN {X 0,Y 380.36,Z 501.902,A -85,B 0,C 180,E1 -20823.845,E2 -20823.845} C_VEL
LIN {X 0,Y 381.961,Z 490.686,A -85,B 0,C 180,E1 -20824.8,E2 -20824.8} C_VEL
LIN {X 0,Y 383.456,Z 477.597,A -85,B 0,C 180,E1 -20825.685,E2 -20825.685} C_VEL
LIN {X 0,Y 384.742,Z 463.52,A -85,B 0,C 180,E1 -20826.394,E2 -20826.394} C_VEL
LIN {X 0,Y 385.583,Z 449.997,A -85,B 0,C 180,E1 -20826.869,E2 -20826.869} C_VEL
LIN {X 0,Y 386.289,Z 426.604,A -85,B 0,C 180,E1 -20827.359,E2 -20827.359} C_VEL
LIN {X 0,Y 388.442,Z 357.854,A -85,B 0,C 180,E1 -20828.633,E2 -20828.633} C_VEL
LIN {X 0,Y 385.927,Z 351.917,A -85,B 0,C 180,E1 -20828.99,E2 -20828.99} C_VEL
LIN {X 0,Y 384.245,Z 348.702,A -85,B 0,C 180,E1 -20829.215,E2 -20829.215} C_VEL
LIN {X 0,Y 380.994,Z 344.52,A -85,B 0,C 180,E1 -20829.614,E2 -20829.614} C_VEL
LIN {X 0,Y 371.199,Z 334.605,A -85,B 0,C 180,E1 -20830.805,E2 -20830.805} C_VEL
LIN {X 0,Y 368.219,Z 330.175,A -85,B 0,C 180,E1 -20831.217,E2 -20831.217} C_VEL
LIN {X 0,Y 360.691,Z 316.678,A -85,B 0,C 180,E1 -20832.356,E2 -20832.356} C_VEL
LIN {X 0,Y 359.226,Z 313.736,A -85,B 0,C 180,E1 -20832.612,E2 -20832.612} C_VEL
LIN {X 0,Y 358.9,Z 312.341,A -85,B 0,C 180,E1 -20833.156,E2 -20833.156} C_VEL
LIN {X 0,Y 358.906,Z 312.329,A -85,B 0,C 180,E1 -20836.223,E2 -20836.223} C_VEL
LIN {X 0,Y 358.894,Z 312.334,A -85,B 0,C 180,E1 -20839.905,E2 -20839.905} C_VEL
LIN {X 0,Y 358.942,Z 312.308,A -85,B 0,C 180,E1 -20843.132,E2 -20843.132} C_VEL
LIN {X 0,Y 358.938,Z 312.307,A -85,B 0,C 180,E1 -20845.534,E2 -20845.534} C_VEL
LIN {X 0,Y 358.984,Z 312.318,A -85,B 0,C 180,E1 -20849.515,E2 -20849.515} C_VEL
LIN {X 0,Y 358.948,Z 312.321,A -85,B 0,C 180,E1 -20852.074,E2 -20852.074} C_VEL
LIN {X 0,Y 358.949,Z 312.33,A -85,B 0,C 180,E1 -20854.577,E2 -20854.577} C_VEL
LIN {X 0,Y 358.963,Z 312.316,A -85,B 0,C 180,E1 -20857.029,E2 -20857.029} C_VEL
LIN {X 0,Y 358.989,Z 312.314,A -85,B 0,C 180,E1 -20860.628,E2 -20860.628} C_VEL
LIN {X 0,Y 358.996,Z 312.322,A -85,B 0,C 180,E1 -20864.148,E2 -20864.148} C_VEL
LIN {X 0,Y 359.14,Z 312.304,A -85,B 0,C 180,E1 -20867.612,E2 -20867.612} C_VEL
LIN {X 0,Y 359.167,Z 312.287,A -85,B 0,C 180,E1 -20871.024,E2 -20871.024} C_VEL
LIN {X 0,Y 359.275,Z 312.288,A -85,B 0,C 180,E1 -20874.406,E2 -20874.406} C_VEL
LIN {X 0,Y 359.309,Z 312.266,A -85,B 0,C 180,E1 -20876.647,E2 -20876.647} C_VEL
LIN {X 0,Y 359.295,Z 312.284,A -85,B 0,C 180,E1 -20880,E2 -20880} C_VEL
LIN {X 0,Y 359.312,Z 312.277,A -85,B 0,C 180,E1 -20883.353,E2 -20883.353} C_VEL
LIN {X 0,Y 359.276,Z 312.273,A -85,B 0,C 180,E1 -20886.718,E2 -20886.718} C_VEL
LIN {X 0,Y 359.151,Z 312.301,A -85,B 0,C 180,E1 -20890.109,E2 -20890.109} C_VEL
LIN {X 0,Y 359.11,Z 312.297,A -85,B 0,C 180,E1 -20893.536,E2 -20893.536} C_VEL
LIN {X 0,Y 359.068,Z 312.297,A -85,B 0,C 180,E1 -20897.1,E2 -20897.1} C_VEL
LIN {X 0,Y 359.008,Z 312.32,A -85,B 0,C 180,E1 -20900.56,E2 -20900.56} C_VEL
LIN {X 0,Y 358.944,Z 312.33,A -85,B 0,C 180,E1 -20904.192,E2 -20904.192} C_VEL
LIN {X 0,Y 358.938,Z 312.321,A -85,B 0,C 180,E1 -20906.669,E2 -20906.669} C_VEL
LIN {X 0,Y 358.941,Z 312.329,A -85,B 0,C 180,E1 -20909.2,E2 -20909.2} C_VEL
LIN {X 0,Y 358.94,Z 312.329,A -85,B 0,C 180,E1 -20911.795,E2 -20911.795} C_VEL
LIN {X 0,Y 359.012,Z 312.283,A -85,B 0,C 180,E1 -20915.825,E2 -20915.825} C_VEL
LIN {X 0,Y 358.976,Z 312.329,A -85,B 0,C 180,E1 -20918.7,E2 -20918.7} C_VEL
LIN {X 0,Y 358.935,Z 312.331,A -85,B 0,C 180,E1 -20922.141,E2 -20922.141} C_VEL
LIN {X 0,Y 358.955,Z 312.325,A -85,B 0,C 180,E1 -20925.378,E2 -20925.378} C_VEL
LIN {X 0,Y 358.959,Z 312.331,A -85,B 0,C 180,E1 -20928.441,E2 -20928.441} C_VEL
LIN {X 0,Y 359.005,Z 312.528,A -85,B 0,C 180,E1 -20930.529,E2 -20930.529} C_VEL
LIN {X 0,Y 361.767,Z 322.252,A -85,B 0,C 180,E1 -20933.449,E2 -20933.449} C_VEL
LIN {X 0,Y 364.438,Z 332.966,A -85,B 0,C 180,E1 -20936.461,E2 -20936.461} C_VEL
LIN {X 0,Y 367.134,Z 345.517,A -85,B 0,C 180,E1 -20939.74,E2 -20939.74} C_VEL
LIN {X 0,Y 367.693,Z 348.179,A -85,B 0,C 180,E1 -20940.393,E2 -20940.393} C_VEL
LIN {X 0,Y 371.505,Z 357.092,A -85,B 0,C 180,E1 -20940.988,E2 -20940.988} C_VEL
LIN {X 0,Y 377.204,Z 387.376,A -85,B 0,C 180,E1 -20942.221,E2 -20942.221} C_VEL
LIN {X 0,Y 380.749,Z 411.692,A -85,B 0,C 180,E1 -20943.081,E2 -20943.081} C_VEL
LIN {X 0,Y 379.005,Z 468.272,A -85,B 0,C 180,E1 -20944.152,E2 -20944.152} C_VEL
LIN {X 0,Y 378.174,Z 489.714,A -85,B 0,C 180,E1 -20944.606,E2 -20944.606} C_VEL
LIN {X 0,Y 376.964,Z 504.046,A -85,B 0,C 180,E1 -20945.107,E2 -20945.107} C_VEL
LIN {X 0,Y 375.241,Z 517.297,A -85,B 0,C 180,E1 -20945.757,E2 -20945.757} C_VEL
LIN {X 0,Y 373.502,Z 528.953,A -85,B 0,C 180,E1 -20946.518,E2 -20946.518} C_VEL
LIN {X 0,Y 371.298,Z 541.411,A -85,B 0,C 180,E1 -20947.546,E2 -20947.546} C_VEL
LIN {X 0,Y 368.888,Z 553.962,A -85,B 0,C 180,E1 -20948.856,E2 -20948.856} C_VEL
LIN {X 0,Y 366.608,Z 564.266,A -85,B 0,C 180,E1 -20950.179,E2 -20950.179} C_VEL
LIN {X 0,Y 364.17,Z 574.563,A -85,B 0,C 180,E1 -20951.79,E2 -20951.79} C_VEL
LIN {X 0,Y 362.122,Z 583.099,A -85,B 0,C 180,E1 -20953.426,E2 -20953.426} C_VEL
LIN {X 0,Y 360.236,Z 591.313,A -85,B 0,C 180,E1 -20955.361,E2 -20955.361} C_VEL
LIN {X 0,Y 358.965,Z 597.094,A -85,B 0,C 180,E1 -20957.036,E2 -20957.036} C_VEL
LIN {X 0,Y 357.65,Z 603.29,A -85,B 0,C 180,E1 -20959.28,E2 -20959.28} C_VEL
LIN {X 0,Y 356.998,Z 606.858,A -85,B 0,C 180,E1 -20960.972,E2 -20960.972} C_VEL
LIN {X 0,Y 356.56,Z 610.389,A -85,B 0,C 180,E1 -20963.234,E2 -20963.234} C_VEL
LIN {X 0,Y 356.598,Z 612.53,A -85,B 0,C 180,E1 -20965.285,E2 -20965.285} C_VEL
LIN {X 0,Y 356.555,Z 616.927,A -85,B 0,C 180,E1 -20967.188,E2 -20967.188} C_VEL
LIN {X 0,Y 356.573,Z 619.854,A -85,B 0,C 180,E1 -20968.877,E2 -20968.877} C_VEL
LIN {X 0,Y 356.487,Z 622.329,A -85,B 0,C 180,E1 -20971.129,E2 -20971.129} C_VEL
LIN {X 0,Y 356.379,Z 623.337,A -85,B 0,C 180,E1 -20973.383,E2 -20973.383} C_VEL
LIN {X 0,Y 356.584,Z 622.922,A -85,B 0,C 180,E1 -20975.639,E2 -20975.639} C_VEL
LIN {X 0,Y 356.956,Z 621.1,A -85,B 0,C 180,E1 -20977.898,E2 -20977.898} C_VEL
LIN {X 0,Y 357.945,Z 617.859,A -85,B 0,C 180,E1 -20980.146,E2 -20980.146} C_VEL
LIN {X 0,Y 359.477,Z 613.108,A -85,B 0,C 180,E1 -20982.379,E2 -20982.379} C_VEL
LIN {X 0,Y 360.754,Z 608.629,A -85,B 0,C 180,E1 -20983.991,E2 -20983.991} C_VEL
LIN {X 0,Y 362.926,Z 601.772,A -85,B 0,C 180,E1 -20985.966,E2 -20985.966} C_VEL
LIN {X 0,Y 365.463,Z 593.559,A -85,B 0,C 180,E1 -20987.86,E2 -20987.86} C_VEL
LIN {X 0,Y 367.789,Z 585.051,A -85,B 0,C 180,E1 -20989.471,E2 -20989.471} C_VEL
LIN {X 0,Y 370.673,Z 574.854,A -85,B 0,C 180,E1 -20991.043,E2 -20991.043} C_VEL
LIN {X 0,Y 373.751,Z 562.522,A -85,B 0,C 180,E1 -20992.596,E2 -20992.596} C_VEL
LIN {X 0,Y 376.772,Z 550.018,A -85,B 0,C 180,E1 -20993.853,E2 -20993.853} C_VEL
LIN {X 0,Y 379.257,Z 537.901,A -85,B 0,C 180,E1 -20994.848,E2 -20994.848} C_VEL
LIN {X 0,Y 381.717,Z 524.71,A -85,B 0,C 180,E1 -20995.693,E2 -20995.693} C_VEL
LIN {X 0,Y 383.881,Z 510.661,A -85,B 0,C 180,E1 -20996.387,E2 -20996.387} C_VEL
LIN {X 0,Y 385.707,Z 495.067,A -85,B 0,C 180,E1 -20996.941,E2 -20996.941} C_VEL
LIN {X 0,Y 392.663,Z 413.899,A -85,B 0,C 180,E1 -20999.302,E2 -20999.302} C_VEL
LIN {X 0,Y 391.808,Z 395.547,A -85,B 0,C 180,E1 -21000.265,E2 -21000.265} C_VEL
LIN {X 0,Y 390.155,Z 377.248,A -85,B 0,C 180,E1 -21001.415,E2 -21001.415} C_VEL
LIN {X 0,Y 388.902,Z 368.362,A -85,B 0,C 180,E1 -21002.089,E2 -21002.089} C_VEL
LIN {X 0,Y 385.249,Z 357.691,A -85,B 0,C 180,E1 -21003.386,E2 -21003.386} C_VEL
LIN {X 0,Y 382.001,Z 352.744,A -85,B 0,C 180,E1 -21004.398,E2 -21004.398} C_VEL
LIN {X 0,Y 378.056,Z 345.274,A -85,B 0,C 180,E1 -21006.626,E2 -21006.626} C_VEL
LIN {X 0,Y 374.534,Z 339.186,A -85,B 0,C 180,E1 -21008.985,E2 -21008.985} C_VEL
LIN {X 0,Y 372.557,Z 335.761,A -85,B 0,C 180,E1 -21010.632,E2 -21010.632} C_VEL
LIN {X 0,Y 370.445,Z 331.956,A -85,B 0,C 180,E1 -21012.901,E2 -21012.901} C_VEL
LIN {X 0,Y 368.178,Z 328.711,A -85,B 0,C 180,E1 -21016.3,E2 -21016.3} C_VEL
LIN {X 0,Y 367.69,Z 327.53,A -85,B 0,C 180,E1 -21018.184,E2 -21018.184} C_VEL
LIN {X 0,Y 367.472,Z 327.114,A -85,B 0,C 180,E1 -21019.683,E2 -21019.683} C_VEL
LIN {X 0,Y 367.424,Z 327.349,A -85,B 0,C 180,E1 -21021.411,E2 -21021.411} C_VEL
LIN {X 0,Y 368.148,Z 329.613,A -85,B 0,C 180,E1 -21025.195,E2 -21025.195} C_VEL
LIN {X 0,Y 368.808,Z 331.049,A -85,B 0,C 180,E1 -21026.687,E2 -21026.687} C_VEL
LIN {X 0,Y 370.258,Z 334.57,A -85,B 0,C 180,E1 -21029.284,E2 -21029.284} C_VEL
LIN {X 0,Y 372.087,Z 339.28,A -85,B 0,C 180,E1 -21031.925,E2 -21031.925} C_VEL
LIN {X 0,Y 374.079,Z 345.012,A -85,B 0,C 180,E1 -21034.49,E2 -21034.49} C_VEL
LIN {X 0,Y 375.476,Z 349.092,A -85,B 0,C 180,E1 -21036.034,E2 -21036.034} C_VEL
LIN {X 0,Y 379.604,Z 355.95,A -85,B 0,C 180,E1 -21037.524,E2 -21037.524} C_VEL
LIN {X 0,Y 384.382,Z 364.188,A -85,B 0,C 180,E1 -21039.064,E2 -21039.064} C_VEL
LIN {X 0,Y 390.221,Z 376.266,A -85,B 0,C 180,E1 -21040.831,E2 -21040.831} C_VEL
LIN {X 0,Y 392.366,Z 381.763,A -85,B 0,C 180,E1 -21041.472,E2 -21041.472} C_VEL
LIN {X 0,Y 394.31,Z 395.975,A -85,B 0,C 180,E1 -21042.441,E2 -21042.441} C_VEL
LIN {X 0,Y 394.192,Z 399.09,A -85,B 0,C 180,E1 -21042.559,E2 -21042.559} C_VEL
LIN {X 0,Y 386.002,Z 490.271,A -85,B 0,C 180,E1 -21045.182,E2 -21045.182} C_VEL
LIN {X 0,Y 384.016,Z 505.949,A -85,B 0,C 180,E1 -21045.866,E2 -21045.866} C_VEL
LIN {X 0,Y 381.673,Z 520.896,A -85,B 0,C 180,E1 -21046.761,E2 -21046.761} C_VEL
LIN {X 0,Y 378.89,Z 535.089,A -85,B 0,C 180,E1 -21047.861,E2 -21047.861} C_VEL
LIN {X 0,Y 376.032,Z 547.993,A -85,B 0,C 180,E1 -21049.129,E2 -21049.129} C_VEL
LIN {X 0,Y 373.072,Z 559.708,A -85,B 0,C 180,E1 -21050.544,E2 -21050.544} C_VEL
LIN {X 0,Y 370.264,Z 570.179,A -85,B 0,C 180,E1 -21052.117,E2 -21052.117} C_VEL
LIN {X 0,Y 367.694,Z 578.94,A -85,B 0,C 180,E1 -21053.711,E2 -21053.711} C_VEL
LIN {X 0,Y 364.949,Z 587.432,A -85,B 0,C 180,E1 -21055.597,E2 -21055.597} C_VEL
LIN {X 0,Y 362.837,Z 593.417,A -85,B 0,C 180,E1 -21057.234,E2 -21057.234} C_VEL
LIN {X 0,Y 360.665,Z 599.751,A -85,B 0,C 180,E1 -21059.444,E2 -21059.444} C_VEL
LIN {X 0,Y 359.355,Z 603.394,A -85,B 0,C 180,E1 -21061.117,E2 -21061.117} C_VEL
LIN {X 0,Y 358.12,Z 606.913,A -85,B 0,C 180,E1 -21063.364,E2 -21063.364} C_VEL
LIN {X 0,Y 357.199,Z 608.998,A -85,B 0,C 180,E1 -21065.627,E2 -21065.627} C_VEL
LIN {X 0,Y 356.533,Z 609.675,A -85,B 0,C 180,E1 -21067.904,E2 -21067.904} C_VEL
LIN {X 0,Y 356.3,Z 608.885,A -85,B 0,C 180,E1 -21070.191,E2 -21070.191} C_VEL
LIN {X 0,Y 356.117,Z 606.583,A -85,B 0,C 180,E1 -21072.495,E2 -21072.495} C_VEL
LIN {X 0,Y 356.246,Z 602.716,A -85,B 0,C 180,E1 -21074.809,E2 -21074.809} C_VEL
LIN {X 0,Y 356.436,Z 598.679,A -85,B 0,C 180,E1 -21076.556,E2 -21076.556} C_VEL
LIN {X 0,Y 356.659,Z 593.549,A -85,B 0,C 180,E1 -21078.314,E2 -21078.314} C_VEL
LIN {X 0,Y 357.091,Z 586.107,A -85,B 0,C 180,E1 -21080.345,E2 -21080.345} C_VEL
LIN {X 0,Y 357.591,Z 577.922,A -85,B 0,C 180,E1 -21082.152,E2 -21082.152} C_VEL
LIN {X 0,Y 358.28,Z 568.119,A -85,B 0,C 180,E1 -21083.933,E2 -21083.933} C_VEL
LIN {X 0,Y 359.098,Z 557.248,A -85,B 0,C 180,E1 -21085.552,E2 -21085.552} C_VEL
LIN {X 0,Y 360.11,Z 545.018,A -85,B 0,C 180,E1 -21087.043,E2 -21087.043} C_VEL
LIN {X 0,Y 361.067,Z 531.579,A -85,B 0,C 180,E1 -21088.378,E2 -21088.378} C_VEL
LIN {X 0,Y 361.927,Z 518.234,A -85,B 0,C 180,E1 -21089.434,E2 -21089.434} C_VEL
LIN {X 0,Y 362.82,Z 504.335,A -85,B 0,C 180,E1 -21090.289,E2 -21090.289} C_VEL
LIN {X 0,Y 363.626,Z 489.256,A -85,B 0,C 180,E1 -21090.976,E2 -21090.976} C_VEL
LIN {X 0,Y 364.216,Z 471.151,A -85,B 0,C 180,E1 -21091.524,E2 -21091.524} C_VEL
LIN {X 0,Y 367.016,Z 382.113,A -85,B 0,C 180,E1 -21093.908,E2 -21093.908} C_VEL
LIN {X 0,Y 363.136,Z 347.661,A -85,B 0,C 180,E1 -21095.01,E2 -21095.01} C_VEL
LIN {X 0,Y 362.972,Z 345.254,A -85,B 0,C 180,E1 -21095.112,E2 -21095.112} C_VEL
LIN {X 0,Y 363.604,Z 336.155,A -85,B 0,C 180,E1 -21096.668,E2 -21096.668} C_VEL
LIN {X 0,Y 361.545,Z 325.085,A -85,B 0,C 180,E1 -21098.682,E2 -21098.682} C_VEL
LIN {X 0,Y 358.928,Z 312.333,A -85,B 0,C 180,E1 -21101.053,E2 -21101.053} C_VEL
LIN {X 0,Y 358.939,Z 312.329,A -85,B 0,C 180,E1 -21104.629,E2 -21104.629} C_VEL
LIN {X 0,Y 358.889,Z 312.339,A -85,B 0,C 180,E1 -21108.424,E2 -21108.424} C_VEL
LIN {X 0,Y 358.911,Z 312.331,A -85,B 0,C 180,E1 -21111.351,E2 -21111.351} C_VEL
LIN {X 0,Y 358.915,Z 312.333,A -85,B 0,C 180,E1 -21114.161,E2 -21114.161} C_VEL
LIN {X 0,Y 358.906,Z 312.329,A -85,B 0,C 180,E1 -21117.055,E2 -21117.055} C_VEL
LIN {X 0,Y 358.953,Z 312.328,A -85,B 0,C 180,E1 -21119.51,E2 -21119.51} C_VEL
LIN {X 0,Y 358.957,Z 312.325,A -85,B 0,C 180,E1 -21123.33,E2 -21123.33} C_VEL
LIN {X 0,Y 358.984,Z 312.324,A -85,B 0,C 180,E1 -21127.028,E2 -21127.028} C_VEL
LIN {X 0,Y 359.021,Z 312.319,A -85,B 0,C 180,E1 -21130.627,E2 -21130.627} C_VEL
LIN {X 0,Y 359.068,Z 312.317,A -85,B 0,C 180,E1 -21134.148,E2 -21134.148} C_VEL
LIN {X 0,Y 359.165,Z 312.355,A -85,B 0,C 180,E1 -21137.386,E2 -21137.386} C_VEL
LIN {X 0,Y 361.402,Z 318.275,A -85,B 0,C 180,E1 -21137.644,E2 -21137.644} C_VEL
LIN {X 0,Y 369.506,Z 341.787,A -85,B 0,C 180,E1 -21138.591,E2 -21138.591} C_VEL
LIN {X 0,Y 370.333,Z 345.007,A -85,B 0,C 180,E1 -21138.702,E2 -21138.702} C_VEL
LIN {X 0,Y 367.92,Z 447.474,A -85,B 0,C 180,E1 -21140.685,E2 -21140.685} C_VEL
LIN {X 0,Y 367.329,Z 461.882,A -85,B 0,C 180,E1 -21141.188,E2 -21141.188} C_VEL
LIN {X 0,Y 366.582,Z 475.679,A -85,B 0,C 180,E1 -21141.897,E2 -21141.897} C_VEL
LIN {X 0,Y 365.464,Z 489.46,A -85,B 0,C 180,E1 -21142.841,E2 -21142.841} C_VEL
LIN {X 0,Y 364.404,Z 500.402,A -85,B 0,C 180,E1 -21143.79,E2 -21143.79} C_VEL
LIN {X 0,Y 363.004,Z 511.991,A -85,B 0,C 180,E1 -21145.016,E2 -21145.016} C_VEL
LIN {X 0,Y 361.982,Z 522.533,A -85,B 0,C 180,E1 -21146.392,E2 -21146.392} C_VEL
LIN {X 0,Y 360.605,Z 533.058,A -85,B 0,C 180,E1 -21148.049,E2 -21148.049} C_VEL
LIN {X 0,Y 359.57,Z 541.729,A -85,B 0,C 180,E1 -21149.718,E2 -21149.718} C_VEL
LIN {X 0,Y 358.426,Z 550.085,A -85,B 0,C 180,E1 -21151.677,E2 -21151.677} C_VEL
LIN {X 0,Y 357.964,Z 556.863,A -85,B 0,C 180,E1 -21153.679,E2 -21153.679} C_VEL
LIN {X 0,Y 357.382,Z 562.093,A -85,B 0,C 180,E1 -21155.621,E2 -21155.621} C_VEL
LIN {X 0,Y 356.868,Z 566.681,A -85,B 0,C 180,E1 -21157.894,E2 -21157.894} C_VEL
LIN {X 0,Y 356.729,Z 569.795,A -85,B 0,C 180,E1 -21160.176,E2 -21160.176} C_VEL
LIN {X 0,Y 356.753,Z 571.541,A -85,B 0,C 180,E1 -21162.47,E2 -21162.47} C_VEL
LIN {X 0,Y 356.98,Z 571.939,A -85,B 0,C 180,E1 -21164.775,E2 -21164.775} C_VEL
LIN {X 0,Y 357.47,Z 570.979,A -85,B 0,C 180,E1 -21167.089,E2 -21167.089} C_VEL
LIN {X 0,Y 358.258,Z 568.627,A -85,B 0,C 180,E1 -21169.41,E2 -21169.41} C_VEL
LIN {X 0,Y 359.452,Z 564.795,A -85,B 0,C 180,E1 -21171.727,E2 -21171.727} C_VEL
LIN {X 0,Y 360.613,Z 560.819,A -85,B 0,C 180,E1 -21173.461,E2 -21173.461} C_VEL
LIN {X 0,Y 361.962,Z 555.866,A -85,B 0,C 180,E1 -21175.193,E2 -21175.193} C_VEL
LIN {X 0,Y 363.97,Z 548.673,A -85,B 0,C 180,E1 -21177.194,E2 -21177.194} C_VEL
LIN {X 0,Y 365.868,Z 541.067,A -85,B 0,C 180,E1 -21178.904,E2 -21178.904} C_VEL
LIN {X 0,Y 368.097,Z 531.855,A -85,B 0,C 180,E1 -21180.595,E2 -21180.595} C_VEL
LIN {X 0,Y 370.352,Z 521.607,A -85,B 0,C 180,E1 -21182.132,E2 -21182.132} C_VEL
LIN {X 0,Y 372.579,Z 510.276,A -85,B 0,C 180,E1 -21183.518,E2 -21183.518} C_VEL
LIN {X 0,Y 374.637,Z 498.105,A -85,B 0,C 180,E1 -21184.716,E2 -21184.716} C_VEL
LIN {X 0,Y 376.446,Z 485.327,A -85,B 0,C 180,E1 -21185.713,E2 -21185.713} C_VEL
LIN {X 0,Y 377.839,Z 471.826,A -85,B 0,C 180,E1 -21186.536,E2 -21186.536} C_VEL
LIN {X 0,Y 379.007,Z 457.193,A -85,B 0,C 180,E1 -21187.175,E2 -21187.175} C_VEL
LIN {X 0,Y 379.718,Z 443.384,A -85,B 0,C 180,E1 -21187.564,E2 -21187.564} C_VEL
LIN {X 0,Y 382.363,Z 359.881,A -85,B 0,C 180,E1 -21189.147,E2 -21189.147} C_VEL
LIN {X 0,Y 374.858,Z 343.204,A -85,B 0,C 180,E1 -21190.241,E2 -21190.241} C_VEL
LIN {X 0,Y 368.219,Z 330.175,A -85,B 0,C 180,E1 -21191.217,E2 -21191.217} C_VEL
LIN {X 0,Y 365.996,Z 327.444,A -85,B 0,C 180,E1 -21191.518,E2 -21191.518} C_VEL
LIN {X 0,Y 356.481,Z 321.375,A -85,B 0,C 180,E1 -21192.722,E2 -21192.722} C_VEL
LIN {X 0,Y 354.507,Z 318.509,A -85,B 0,C 180,E1 -21193.023,E2 -21193.023} C_VEL
LIN {X 0,Y 352.218,Z 314.648,A -85,B 0,C 180,E1 -21193.39,E2 -21193.39} C_VEL
LIN {X 0,Y 351.964,Z 313.722,A -85,B 0,C 180,E1 -21193.623,E2 -21193.623} C_VEL
LIN {X 0,Y 351.871,Z 313.204,A -85,B 0,C 180,E1 -21193.814,E2 -21193.814} C_VEL
LIN {X 0,Y 351.857,Z 313.213,A -85,B 0,C 180,E1 -21197.434,E2 -21197.434} C_VEL
LIN {X 0,Y 351.853,Z 313.213,A -85,B 0,C 180,E1 -21200.925,E2 -21200.925} C_VEL
LIN {X 0,Y 351.888,Z 313.183,A -85,B 0,C 180,E1 -21203.333,E2 -21203.333} C_VEL
LIN {X 0,Y 351.874,Z 313.21,A -85,B 0,C 180,E1 -21206.72,E2 -21206.72} C_VEL
LIN {X 0,Y 351.906,Z 313.206,A -85,B 0,C 180,E1 -21210.158,E2 -21210.158} C_VEL
LIN {X 0,Y 351.908,Z 313.2,A -85,B 0,C 180,E1 -21213.589,E2 -21213.589} C_VEL
LIN {X 0,Y 351.957,Z 313.188,A -85,B 0,C 180,E1 -21216.545,E2 -21216.545} C_VEL
LIN {X 0,Y 351.937,Z 313.196,A -85,B 0,C 180,E1 -21220.224,E2 -21220.224} C_VEL
LIN {X 0,Y 351.964,Z 313.2,A -85,B 0,C 180,E1 -21223.822,E2 -21223.822} C_VEL
LIN {X 0,Y 352.09,Z 313.178,A -85,B 0,C 180,E1 -21227.36,E2 -21227.36} C_VEL
LIN {X 0,Y 352.133,Z 313.163,A -85,B 0,C 180,E1 -21230.844,E2 -21230.844} C_VEL
LIN {X 0,Y 352.236,Z 313.165,A -85,B 0,C 180,E1 -21234.294,E2 -21234.294} C_VEL
LIN {X 0,Y 352.294,Z 313.151,A -85,B 0,C 180,E1 -21237.721,E2 -21237.721} C_VEL
LIN {X 0,Y 352.24,Z 313.149,A -85,B 0,C 180,E1 -21241.139,E2 -21241.139} C_VEL
LIN {X 0,Y 352.309,Z 313.157,A -85,B 0,C 180,E1 -21244.561,E2 -21244.561} C_VEL
LIN {X 0,Y 352.226,Z 313.15,A -85,B 0,C 180,E1 -21246.853,E2 -21246.853} C_VEL
LIN {X 0,Y 352.112,Z 313.179,A -85,B 0,C 180,E1 -21250.314,E2 -21250.314} C_VEL
LIN {X 0,Y 352.046,Z 313.18,A -85,B 0,C 180,E1 -21253.813,E2 -21253.813} C_VEL
LIN {X 0,Y 351.997,Z 313.177,A -85,B 0,C 180,E1 -21257.367,E2 -21257.367} C_VEL
LIN {X 0,Y 351.939,Z 313.194,A -85,B 0,C 180,E1 -21260.992,E2 -21260.992} C_VEL
LIN {X 0,Y 351.925,Z 313.202,A -85,B 0,C 180,E1 -21263.725,E2 -21263.725} C_VEL
LIN {X 0,Y 351.891,Z 313.202,A -85,B 0,C 180,E1 -21267.246,E2 -21267.246} C_VEL
LIN {X 0,Y 351.911,Z 313.2,A -85,B 0,C 180,E1 -21269.841,E2 -21269.841} C_VEL
LIN {X 0,Y 351.893,Z 313.191,A -85,B 0,C 180,E1 -21273.872,E2 -21273.872} C_VEL
LIN {X 0,Y 351.971,Z 313.175,A -85,B 0,C 180,E1 -21277.254,E2 -21277.254} C_VEL
LIN {X 0,Y 351.909,Z 313.206,A -85,B 0,C 180,E1 -21281.059,E2 -21281.059} C_VEL
LIN {X 0,Y 351.915,Z 313.208,A -85,B 0,C 180,E1 -21284.236,E2 -21284.236} C_VEL
LIN {X 0,Y 351.91,Z 313.203,A -85,B 0,C 180,E1 -21287.43,E2 -21287.43} C_VEL
LIN {X 0,Y 351.964,Z 313.38,A -85,B 0,C 180,E1 -21289.787,E2 -21289.787} C_VEL
LIN {X 0,Y 354.9,Z 323.801,A -85,B 0,C 180,E1 -21293.024,E2 -21293.024} C_VEL
LIN {X 0,Y 357.59,Z 334.454,A -85,B 0,C 180,E1 -21296.084,E2 -21296.084} C_VEL
LIN {X 0,Y 360.076,Z 345.889,A -85,B 0,C 180,E1 -21299.169,E2 -21299.169} C_VEL
LIN {X 0,Y 360.445,Z 347.718,A -85,B 0,C 180,E1 -21299.609,E2 -21299.609} C_VEL
LIN {X 0,Y 365.905,Z 360.115,A -85,B 0,C 180,E1 -21300.484,E2 -21300.484} C_VEL
LIN {X 0,Y 371.374,Z 389.795,A -85,B 0,C 180,E1 -21301.715,E2 -21301.715} C_VEL
LIN {X 0,Y 374.712,Z 413.013,A -85,B 0,C 180,E1 -21302.555,E2 -21302.555} C_VEL
LIN {X 0,Y 372.212,Z 486.499,A -85,B 0,C 180,E1 -21303.982,E2 -21303.982} C_VEL
LIN {X 0,Y 371.097,Z 500.982,A -85,B 0,C 180,E1 -21304.461,E2 -21304.461} C_VEL
LIN {X 0,Y 369.36,Z 514.901,A -85,B 0,C 180,E1 -21305.121,E2 -21305.121} C_VEL
LIN {X 0,Y 367.308,Z 527.869,A -85,B 0,C 180,E1 -21305.948,E2 -21305.948} C_VEL
LIN {X 0,Y 364.931,Z 540.995,A -85,B 0,C 180,E1 -21307.04,E2 -21307.04} C_VEL
LIN {X 0,Y 362.669,Z 552.486,A -85,B 0,C 180,E1 -21308.25,E2 -21308.25} C_VEL
LIN {X 0,Y 360.383,Z 562.491,A -85,B 0,C 180,E1 -21309.525,E2 -21309.525} C_VEL
LIN {X 0,Y 357.783,Z 573.016,A -85,B 0,C 180,E1 -21311.157,E2 -21311.157} C_VEL
LIN {X 0,Y 355.612,Z 581.736,A -85,B 0,C 180,E1 -21312.818,E2 -21312.818} C_VEL
LIN {X 0,Y 353.608,Z 590.143,A -85,B 0,C 180,E1 -21314.787,E2 -21314.787} C_VEL
LIN {X 0,Y 352.016,Z 596.949,A -85,B 0,C 180,E1 -21316.775,E2 -21316.775} C_VEL
LIN {X 0,Y 350.958,Z 601.663,A -85,B 0,C 180,E1 -21318.491,E2 -21318.491} C_VEL
LIN {X 0,Y 349.972,Z 606.601,A -85,B 0,C 180,E1 -21320.789,E2 -21320.789} C_VEL
LIN {X 0,Y 349.466,Z 610.08,A -85,B 0,C 180,E1 -21323.096,E2 -21323.096} C_VEL
LIN {X 0,Y 349.522,Z 612.287,A -85,B 0,C 180,E1 -21325.405,E2 -21325.405} C_VEL
LIN {X 0,Y 349.496,Z 616.295,A -85,B 0,C 180,E1 -21327.131,E2 -21327.131} C_VEL
LIN {X 0,Y 349.507,Z 619.317,A -85,B 0,C 180,E1 -21328.854,E2 -21328.854} C_VEL
LIN {X 0,Y 349.409,Z 621.981,A -85,B 0,C 180,E1 -21331.151,E2 -21331.151} C_VEL
LIN {X 0,Y 349.301,Z 623.141,A -85,B 0,C 180,E1 -21333.452,E2 -21333.452} C_VEL
LIN {X 0,Y 349.494,Z 622.875,A -85,B 0,C 180,E1 -21335.754,E2 -21335.754} C_VEL
LIN {X 0,Y 349.902,Z 621.21,A -85,B 0,C 180,E1 -21338.058,E2 -21338.058} C_VEL
LIN {X 0,Y 350.969,Z 618.127,A -85,B 0,C 180,E1 -21340.35,E2 -21340.35} C_VEL
LIN {X 0,Y 352.545,Z 613.564,A -85,B 0,C 180,E1 -21342.627,E2 -21342.627} C_VEL
LIN {X 0,Y 353.961,Z 609.089,A -85,B 0,C 180,E1 -21344.323,E2 -21344.323} C_VEL
LIN {X 0,Y 356.153,Z 602.623,A -85,B 0,C 180,E1 -21346.278,E2 -21346.278} C_VEL
LIN {X 0,Y 358.804,Z 594.628,A -85,B 0,C 180,E1 -21348.203,E2 -21348.203} C_VEL
LIN {X 0,Y 361.233,Z 586.403,A -85,B 0,C 180,E1 -21349.839,E2 -21349.839} C_VEL
LIN {X 0,Y 364.21,Z 576.548,A -85,B 0,C 180,E1 -21351.435,E2 -21351.435} C_VEL
LIN {X 0,Y 367.455,Z 564.723,A -85,B 0,C 180,E1 -21353.005,E2 -21353.005} C_VEL
LIN {X 0,Y 370.5,Z 552.697,A -85,B 0,C 180,E1 -21354.282,E2 -21354.282} C_VEL
LIN {X 0,Y 373.429,Z 539.622,A -85,B 0,C 180,E1 -21355.411,E2 -21355.411} C_VEL
LIN {X 0,Y 375.962,Z 527.016,A -85,B 0,C 180,E1 -21356.265,E2 -21356.265} C_VEL
LIN {X 0,Y 378.181,Z 513.644,A -85,B 0,C 180,E1 -21356.979,E2 -21356.979} C_VEL
LIN {X 0,Y 380.222,Z 498.278,A -85,B 0,C 180,E1 -21357.574,E2 -21357.574} C_VEL
LIN {X 0,Y 387.802,Z 415.04,A -85,B 0,C 180,E1 -21360.047,E2 -21360.047} C_VEL
LIN {X 0,Y 387.041,Z 396.372,A -85,B 0,C 180,E1 -21361.063,E2 -21361.063} C_VEL
LIN {X 0,Y 385.597,Z 379.006,A -85,B 0,C 180,E1 -21362.196,E2 -21362.196} C_VEL
LIN {X 0,Y 384.699,Z 372.156,A -85,B 0,C 180,E1 -21362.729,E2 -21362.729} C_VEL
LIN {X 0,Y 381.747,Z 363.028,A -85,B 0,C 180,E1 -21363.858,E2 -21363.858} C_VEL
LIN {X 0,Y 376.512,Z 355.177,A -85,B 0,C 180,E1 -21365.588,E2 -21365.588} C_VEL
LIN {X 0,Y 374.409,Z 351.982,A -85,B 0,C 180,E1 -21366.443,E2 -21366.443} C_VEL
LIN {X 0,Y 371.314,Z 346.321,A -85,B 0,C 180,E1 -21368.502,E2 -21368.502} C_VEL
LIN {X 0,Y 368.71,Z 341.908,A -85,B 0,C 180,E1 -21370.546,E2 -21370.546} C_VEL
LIN {X 0,Y 366.039,Z 337.33,A -85,B 0,C 180,E1 -21373.351,E2 -21373.351} C_VEL
LIN {X 0,Y 363.858,Z 334.027,A -85,B 0,C 180,E1 -21377.017,E2 -21377.017} C_VEL
LIN {X 0,Y 363.403,Z 333.033,A -85,B 0,C 180,E1 -21379.055,E2 -21379.055} C_VEL
LIN {X 0,Y 363.229,Z 332.916,A -85,B 0,C 180,E1 -21380.479,E2 -21380.479} C_VEL
LIN {X 0,Y 363.148,Z 333.394,A -85,B 0,C 180,E1 -21382.265,E2 -21382.265} C_VEL
LIN {X 0,Y 364.076,Z 335.992,A -85,B 0,C 180,E1 -21386.087,E2 -21386.087} C_VEL
LIN {X 0,Y 365.768,Z 340.386,A -85,B 0,C 180,E1 -21389.517,E2 -21389.517} C_VEL
LIN {X 0,Y 367.015,Z 343.777,A -85,B 0,C 180,E1 -21391.502,E2 -21391.502} C_VEL
LIN {X 0,Y 368.959,Z 349.452,A -85,B 0,C 180,E1 -21394.11,E2 -21394.11} C_VEL
LIN {X 0,Y 373.237,Z 356.201,A -85,B 0,C 180,E1 -21395.889,E2 -21395.889} C_VEL
LIN {X 0,Y 376.71,Z 362.109,A -85,B 0,C 180,E1 -21397.182,E2 -21397.182} C_VEL
LIN {X 0,Y 380.932,Z 369.679,A -85,B 0,C 180,E1 -21398.62,E2 -21398.62} C_VEL
LIN {X 0,Y 386.269,Z 381.023,A -85,B 0,C 180,E1 -21400.316,E2 -21400.316} C_VEL
LIN {X 0,Y 387.935,Z 385.397,A -85,B 0,C 180,E1 -21400.851,E2 -21400.851} C_VEL
LIN {X 0,Y 389.561,Z 398.43,A -85,B 0,C 180,E1 -21401.757,E2 -21401.757} C_VEL
LIN {X 0,Y 380.816,Z 490.78,A -85,B 0,C 180,E1 -21404.463,E2 -21404.463} C_VEL
LIN {X 0,Y 378.785,Z 505.921,A -85,B 0,C 180,E1 -21405.133,E2 -21405.133} C_VEL
LIN {X 0,Y 376.434,Z 520.329,A -85,B 0,C 180,E1 -21406.001,E2 -21406.001} C_VEL
LIN {X 0,Y 373.775,Z 533.505,A -85,B 0,C 180,E1 -21407.004,E2 -21407.004} C_VEL
LIN {X 0,Y 370.724,Z 546.661,A -85,B 0,C 180,E1 -21408.281,E2 -21408.281} C_VEL
LIN {X 0,Y 367.576,Z 558.62,A -85,B 0,C 180,E1 -21409.709,E2 -21409.709} C_VEL
LIN {X 0,Y 364.789,Z 568.506,A -85,B 0,C 180,E1 -21411.164,E2 -21411.164} C_VEL
LIN {X 0,Y 362.064,Z 577.562,A -85,B 0,C 180,E1 -21412.776,E2 -21412.776} C_VEL
LIN {X 0,Y 359.198,Z 586.086,A -85,B 0,C 180,E1 -21414.627,E2 -21414.627} C_VEL
LIN {X 0,Y 356.451,Z 593.437,A -85,B 0,C 180,E1 -21416.62,E2 -21416.62} C_VEL
LIN {X 0,Y 354.123,Z 599.783,A -85,B 0,C 180,E1 -21418.867,E2 -21418.867} C_VEL
LIN {X 0,Y 352.273,Z 604.516,A -85,B 0,C 180,E1 -21421.139,E2 -21421.139} C_VEL
LIN {X 0,Y 351.04,Z 607.697,A -85,B 0,C 180,E1 -21423.432,E2 -21423.432} C_VEL
LIN {X 0,Y 350.052,Z 609.445,A -85,B 0,C 180,E1 -21425.742,E2 -21425.742} C_VEL
LIN {X 0,Y 349.425,Z 609.776,A -85,B 0,C 180,E1 -21428.066,E2 -21428.066} C_VEL
LIN {X 0,Y 349.177,Z 608.667,A -85,B 0,C 180,E1 -21430.401,E2 -21430.401} C_VEL
LIN {X 0,Y 349.027,Z 606.068,A -85,B 0,C 180,E1 -21432.753,E2 -21432.753} C_VEL
LIN {X 0,Y 349.148,Z 603.06,A -85,B 0,C 180,E1 -21434.523,E2 -21434.523} C_VEL
LIN {X 0,Y 349.342,Z 599.092,A -85,B 0,C 180,E1 -21436.302,E2 -21436.302} C_VEL
LIN {X 0,Y 349.541,Z 594.023,A -85,B 0,C 180,E1 -21438.096,E2 -21438.096} C_VEL
LIN {X 0,Y 349.965,Z 586.529,A -85,B 0,C 180,E1 -21440.197,E2 -21440.197} C_VEL
LIN {X 0,Y 350.449,Z 578.556,A -85,B 0,C 180,E1 -21442.009,E2 -21442.009} C_VEL
LIN {X 0,Y 351.141,Z 568.859,A -85,B 0,C 180,E1 -21443.825,E2 -21443.825} C_VEL
LIN {X 0,Y 351.971,Z 558.069,A -85,B 0,C 180,E1 -21445.49,E2 -21445.49} C_VEL
LIN {X 0,Y 352.92,Z 546.254,A -85,B 0,C 180,E1 -21446.981,E2 -21446.981} C_VEL
LIN {X 0,Y 353.91,Z 532.846,A -85,B 0,C 180,E1 -21448.359,E2 -21448.359} C_VEL
LIN {X 0,Y 354.846,Z 519.121,A -85,B 0,C 180,E1 -21449.489,E2 -21449.489} C_VEL
LIN {X 0,Y 355.762,Z 504.443,A -85,B 0,C 180,E1 -21450.415,E2 -21450.415} C_VEL
LIN {X 0,Y 356.54,Z 490.148,A -85,B 0,C 180,E1 -21451.085,E2 -21451.085} C_VEL
LIN {X 0,Y 357.119,Z 473.885,A -85,B 0,C 180,E1 -21451.605,E2 -21451.605} C_VEL
LIN {X 0,Y 360.08,Z 383.02,A -85,B 0,C 180,E1 -21454.109,E2 -21454.109} C_VEL
LIN {X 0,Y 356.161,Z 347.781,A -85,B 0,C 180,E1 -21455.262,E2 -21455.262} C_VEL
LIN {X 0,Y 356.022,Z 345.376,A -85,B 0,C 180,E1 -21455.367,E2 -21455.367} C_VEL
LIN {X 0,Y 356.553,Z 336.779,A -85,B 0,C 180,E1 -21456.85,E2 -21456.85} C_VEL
LIN {X 0,Y 353.867,Z 322.66,A -85,B 0,C 180,E1 -21459.466,E2 -21459.466} C_VEL
LIN {X 0,Y 351.899,Z 313.208,A -85,B 0,C 180,E1 -21461.268,E2 -21461.268} C_VEL
LIN {X 0,Y 351.88,Z 313.213,A -85,B 0,C 180,E1 -21464.222,E2 -21464.222} C_VEL
LIN {X 0,Y 351.851,Z 313.212,A -85,B 0,C 180,E1 -21467.44,E2 -21467.44} C_VEL
LIN {X 0,Y 351.862,Z 313.21,A -85,B 0,C 180,E1 -21470.929,E2 -21470.929} C_VEL
LIN {X 0,Y 351.886,Z 313.207,A -85,B 0,C 180,E1 -21473.33,E2 -21473.33} C_VEL
LIN {X 0,Y 351.871,Z 313.207,A -85,B 0,C 180,E1 -21476.727,E2 -21476.727} C_VEL
LIN {X 0,Y 351.889,Z 313.21,A -85,B 0,C 180,E1 -21480.154,E2 -21480.154} C_VEL
LIN {X 0,Y 351.949,Z 313.203,A -85,B 0,C 180,E1 -21484.031,E2 -21484.031} C_VEL
LIN {X 0,Y 351.98,Z 313.198,A -85,B 0,C 180,E1 -21486.544,E2 -21486.544} C_VEL
LIN {X 0,Y 351.968,Z 313.201,A -85,B 0,C 180,E1 -21490.223,E2 -21490.223} C_VEL
LIN {X 0,Y 352.027,Z 313.193,A -85,B 0,C 180,E1 -21493.823,E2 -21493.823} C_VEL
LIN {X 0,Y 352.11,Z 313.182,A -85,B 0,C 180,E1 -21496.961,E2 -21496.961} C_VEL
LIN {X 0,Y 354.407,Z 319.139,A -85,B 0,C 180,E1 -21497.24,E2 -21497.24} C_VEL
LIN {X 0,Y 362.066,Z 340.815,A -85,B 0,C 180,E1 -21498.153,E2 -21498.153} C_VEL
LIN {X 0,Y 363.63,Z 345.804,A -85,B 0,C 180,E1 -21498.346,E2 -21498.346} C_VEL
LIN {X 0,Y 361.191,Z 447.123,A -85,B 0,C 180,E1 -21500.334,E2 -21500.334} C_VEL
LIN {X 0,Y 360.586,Z 461.819,A -85,B 0,C 180,E1 -21500.846,E2 -21500.846} C_VEL
LIN {X 0,Y 359.846,Z 475.182,A -85,B 0,C 180,E1 -21501.532,E2 -21501.532} C_VEL
LIN {X 0,Y 358.76,Z 488.289,A -85,B 0,C 180,E1 -21502.424,E2 -21502.424} C_VEL
LIN {X 0,Y 357.723,Z 499.516,A -85,B 0,C 180,E1 -21503.392,E2 -21503.392} C_VEL
LIN {X 0,Y 356.23,Z 511.344,A -85,B 0,C 180,E1 -21504.638,E2 -21504.638} C_VEL
LIN {X 0,Y 355.126,Z 522.071,A -85,B 0,C 180,E1 -21506.039,E2 -21506.039} C_VEL
LIN {X 0,Y 353.961,Z 531.111,A -85,B 0,C 180,E1 -21507.445,E2 -21507.445} C_VEL
LIN {X 0,Y 352.744,Z 540.192,A -85,B 0,C 180,E1 -21509.144,E2 -21509.144} C_VEL
LIN {X 0,Y 351.762,Z 547.76,A -85,B 0,C 180,E1 -21510.853,E2 -21510.853} C_VEL
LIN {X 0,Y 351.207,Z 553.064,A -85,B 0,C 180,E1 -21512.283,E2 -21512.283} C_VEL
LIN {X 0,Y 350.764,Z 558.423,A -85,B 0,C 180,E1 -21514.004,E2 -21514.004} C_VEL
LIN {X 0,Y 350.115,Z 564.11,A -85,B 0,C 180,E1 -21516.314,E2 -21516.314} C_VEL
LIN {X 0,Y 349.755,Z 567.343,A -85,B 0,C 180,E1 -21518.056,E2 -21518.056} C_VEL
LIN {X 0,Y 349.662,Z 570.365,A -85,B 0,C 180,E1 -21520.384,E2 -21520.384} C_VEL
LIN {X 0,Y 349.681,Z 572.027,A -85,B 0,C 180,E1 -21522.726,E2 -21522.726} C_VEL
LIN {X 0,Y 349.968,Z 572.338,A -85,B 0,C 180,E1 -21525.078,E2 -21525.078} C_VEL
LIN {X 0,Y 350.48,Z 571.291,A -85,B 0,C 180,E1 -21527.441,E2 -21527.441} C_VEL
LIN {X 0,Y 351.367,Z 568.846,A -85,B 0,C 180,E1 -21529.806,E2 -21529.806} C_VEL
LIN {X 0,Y 352.637,Z 564.877,A -85,B 0,C 180,E1 -21532.169,E2 -21532.169} C_VEL
LIN {X 0,Y 354.301,Z 559.257,A -85,B 0,C 180,E1 -21534.526,E2 -21534.526} C_VEL
LIN {X 0,Y 356.136,Z 552.84,A -85,B 0,C 180,E1 -21536.576,E2 -21536.576} C_VEL
LIN {X 0,Y 358.055,Z 546.019,A -85,B 0,C 180,E1 -21538.32,E2 -21538.32} C_VEL
LIN {X 0,Y 360.172,Z 537.791,A -85,B 0,C 180,E1 -21540.047,E2 -21540.047} C_VEL
LIN {X 0,Y 362.442,Z 528.54,A -85,B 0,C 180,E1 -21541.637,E2 -21541.637} C_VEL
LIN {X 0,Y 364.819,Z 517.648,A -85,B 0,C 180,E1 -21543.171,E2 -21543.171} C_VEL
LIN {X 0,Y 366.947,Z 506.645,A -85,B 0,C 180,E1 -21544.433,E2 -21544.433} C_VEL
LIN {X 0,Y 368.939,Z 494.855,A -85,B 0,C 180,E1 -21545.529,E2 -21545.529} C_VEL
LIN {X 0,Y 370.745,Z 481.492,A -85,B 0,C 180,E1 -21546.518,E2 -21546.518} C_VEL
LIN {X 0,Y 372.005,Z 468.653,A -85,B 0,C 180,E1 -21547.249,E2 -21547.249} C_VEL
LIN {X 0,Y 373.115,Z 453.968,A -85,B 0,C 180,E1 -21547.837,E2 -21547.837} C_VEL
LIN {X 0,Y 373.762,Z 438.032,A -85,B 0,C 180,E1 -21548.227,E2 -21548.227} C_VEL
LIN {X 0,Y 376.269,Z 361.834,A -85,B 0,C 180,E1 -21549.684,E2 -21549.684} C_VEL
LIN {X 0,Y 368.296,Z 344.299,A -85,B 0,C 180,E1 -21550.882,E2 -21550.882} C_VEL
LIN {X 0,Y 359.615,Z 327.704,A -85,B 0,C 180,E1 -21552.212,E2 -21552.212} C_VEL
LIN {X 0,Y 354.507,Z 318.509,A -85,B 0,C 180,E1 -21553.023,E2 -21553.023} C_VEL
LIN {X 0,Y 352.973,Z 316.186,A -85,B 0,C 180,E1 -21553.308,E2 -21553.308} C_VEL
LIN {X 0,Y 350.639,Z 314.595,A -85,B 0,C 180,E1 -21553.784,E2 -21553.784} C_VEL
LIN {X 0,Y 347.925,Z 313.923,A -85,B 0,C 180,E1 -21554.447,E2 -21554.447} C_VEL
LIN {X 0,Y 345.472,Z 313.992,A -85,B 0,C 180,E1 -21555.324,E2 -21555.324} C_VEL
LIN {X 0,Y 344.782,Z 314.085,A -85,B 0,C 180,E1 -21556.034,E2 -21556.034} C_VEL
LIN {X 0,Y 344.794,Z 314.094,A -85,B 0,C 180,E1 -21559.453,E2 -21559.453} C_VEL
LIN {X 0,Y 344.831,Z 314.078,A -85,B 0,C 180,E1 -21562.455,E2 -21562.455} C_VEL
LIN {X 0,Y 344.823,Z 314.061,A -85,B 0,C 180,E1 -21565.336,E2 -21565.336} C_VEL
LIN {X 0,Y 344.851,Z 314.079,A -85,B 0,C 180,E1 -21568.542,E2 -21568.542} C_VEL
LIN {X 0,Y 344.875,Z 314.073,A -85,B 0,C 180,E1 -21572.152,E2 -21572.152} C_VEL
LIN {X 0,Y 344.872,Z 314.073,A -85,B 0,C 180,E1 -21576.05,E2 -21576.05} C_VEL
LIN {X 0,Y 344.91,Z 314.074,A -85,B 0,C 180,E1 -21579.804,E2 -21579.804} C_VEL
LIN {X 0,Y 344.926,Z 314.08,A -85,B 0,C 180,E1 -21583.483,E2 -21583.483} C_VEL
LIN {X 0,Y 345.079,Z 314.048,A -85,B 0,C 180,E1 -21587.098,E2 -21587.098} C_VEL
LIN {X 0,Y 345.074,Z 314.043,A -85,B 0,C 180,E1 -21590.655,E2 -21590.655} C_VEL
LIN {X 0,Y 345.212,Z 314.04,A -85,B 0,C 180,E1 -21594.177,E2 -21594.177} C_VEL
LIN {X 0,Y 345.255,Z 314.026,A -85,B 0,C 180,E1 -21597.675,E2 -21597.675} C_VEL
LIN {X 0,Y 345.215,Z 314.023,A -85,B 0,C 180,E1 -21601.163,E2 -21601.163} C_VEL
LIN {X 0,Y 345.265,Z 314.035,A -85,B 0,C 180,E1 -21604.655,E2 -21604.655} C_VEL
LIN {X 0,Y 345.187,Z 314.025,A -85,B 0,C 180,E1 -21606.993,E2 -21606.993} C_VEL
LIN {X 0,Y 345.055,Z 314.059,A -85,B 0,C 180,E1 -21610.527,E2 -21610.527} C_VEL
LIN {X 0,Y 345.066,Z 314.04,A -85,B 0,C 180,E1 -21613.023,E2 -21613.023} C_VEL
LIN {X 0,Y 344.961,Z 314.053,A -85,B 0,C 180,E1 -21617.394,E2 -21617.394} C_VEL
LIN {X 0,Y 344.885,Z 314.07,A -85,B 0,C 180,E1 -21621.443,E2 -21621.443} C_VEL
LIN {X 0,Y 344.849,Z 314.082,A -85,B 0,C 180,E1 -21625.248,E2 -21625.248} C_VEL
LIN {X 0,Y 344.864,Z 314.082,A -85,B 0,C 180,E1 -21629.174,E2 -21629.174} C_VEL
LIN {X 0,Y 344.844,Z 314.086,A -85,B 0,C 180,E1 -21631.878,E2 -21631.878} C_VEL
LIN {X 0,Y 344.881,Z 314.042,A -85,B 0,C 180,E1 -21635.676,E2 -21635.676} C_VEL
LIN {X 0,Y 344.86,Z 314.085,A -85,B 0,C 180,E1 -21639.024,E2 -21639.024} C_VEL
LIN {X 0,Y 344.85,Z 314.086,A -85,B 0,C 180,E1 -21642.089,E2 -21642.089} C_VEL
LIN {X 0,Y 344.844,Z 314.082,A -85,B 0,C 180,E1 -21645.31,E2 -21645.31} C_VEL
LIN {X 0,Y 344.902,Z 314.204,A -85,B 0,C 180,E1 -21648.993,E2 -21648.993} C_VEL
LIN {X 0,Y 348.101,Z 325.38,A -85,B 0,C 180,E1 -21652.596,E2 -21652.596} C_VEL
LIN {X 0,Y 351.031,Z 337.105,A -85,B 0,C 180,E1 -21656.037,E2 -21656.037} C_VEL
LIN {X 0,Y 353.141,Z 347.055,A -85,B 0,C 180,E1 -21658.769,E2 -21658.769} C_VEL
LIN {X 0,Y 360.293,Z 362.972,A -85,B 0,C 180,E1 -21659.956,E2 -21659.956} C_VEL
LIN {X 0,Y 365.507,Z 391.925,A -85,B 0,C 180,E1 -21661.18,E2 -21661.18} C_VEL
LIN {X 0,Y 368.662,Z 414.436,A -85,B 0,C 180,E1 -21662.009,E2 -21662.009} C_VEL
